TRIGGER WHEN DISTANCE=1 DELAY=-1 DO Schrittmerker_R1Place(10692,10691,FPlace_R1_L6_S4_Check,XPlace_R1_L6_S4_Check) PRIO=-1
;FOLD PTP Place_R1_L6_S4_Check Vel=12 % PPlace_R1_L6_S4_Check Tool[1]:Upper Gripper Base[1]:Rack1;%{PE}%R8.3.21,%MKUKATPBASIS,%CMOVE,%VPTP,%P 1:PTP, 2:Place_R1_L6_S4_Check, 3:, 5:12, 7:PPlace_R1_L6_S4_Check
$BWDSTART=FALSE
PDAT_ACT= PPPlace_R1_L6_S4_Check
FDAT_ACT= FPlace_R1_L6_S4_Check
BAS(#PTP_PARAMS,12)
PTP XPlace_R1_L6_S4_Check
;ENDFOLD

;***************************************************
;FOLD Pruefe Platz frei
IF (DetectPart(CHECK_SHELF,PLACE)==OCCUPIED) THEN
  UP_Rueckzug_R1Place( )
  RETURN
ENDIF
;ENDFOLD
;***************************************************

TRIGGER WHEN DISTANCE=1 DELAY=-1 DO Schrittmerker_R1Place(10693,10692,FPlace_R1_L6_S4_VP3,XPlace_R1_L6_S4_VP3) PRIO=-1
;FOLD LIN Place_R1_L6_S4_VP3 CONT Vel=0.5 m/s LPlace_R1_L6_S4_VP3 Tool[1]:Upper Gripper Base[1]:Rack1;%{PE}%R8.3.21,%MKUKATPBASIS,%CMOVE,%VLIN,%P 1:LIN, 2:Place_R1_L6_S4_VP3, 3:C_DIS C_DIS, 5:0.5, 7:LPlace_R1_L6_S4_VP3
$BWDSTART=FALSE
LDAT_ACT= LLPlace_R1_L6_S4_VP3
FDAT_ACT= FPlace_R1_L6_S4_VP3
BAS(#CP_PARAMS,0.5)
LIN XPlace_R1_L6_S4_VP3 C_DIS C_DIS
;ENDFOLD
TRIGGER WHEN DISTANCE=1 DELAY=-1 DO Schrittmerker_R1Place(10694,10693,FPlace_R1_L6_S4_VP4,XPlace_R1_L6_S4_VP4) PRIO=-1
;FOLD LIN Place_R1_L6_S4_VP4 CONT Vel=0.5 m/s LPlace_R1_L6_S4_VP4 Tool[1]:Upper Gripper Base[1]:Rack1;%{PE}%R8.3.21,%MKUKATPBASIS,%CMOVE,%VLIN,%P 1:LIN, 2:Place_R1_L6_S4_VP4, 3:C_DIS C_DIS, 5:0.5, 7:LPlace_R1_L6_S4_VP4
$BWDSTART=FALSE
LDAT_ACT= LLPlace_R1_L6_S4_VP4
FDAT_ACT= FPlace_R1_L6_S4_VP4
BAS(#CP_PARAMS,0.5)
LIN XPlace_R1_L6_S4_VP4 C_DIS C_DIS
;ENDFOLD
TRIGGER WHEN DISTANCE=1 DELAY=-1 DO Schrittmerker_R1Place(10695,10694,FPlace_R1_L6_S4_VP5,XPlace_R1_L6_S4_VP5) PRIO=-1
;FOLD LIN Place_R1_L6_S4_VP5 CONT Vel=0.5 m/s LPlace_R1_L6_S4_VP5 Tool[1]:Upper Gripper Base[1]:Rack1;%{PE}%R8.3.21,%MKUKATPBASIS,%CMOVE,%VLIN,%P 1:LIN, 2:Place_R1_L6_S4_VP5, 3:C_DIS C_DIS, 5:0.5, 7:LPlace_R1_L6_S4_VP5
$BWDSTART=FALSE
LDAT_ACT= LLPlace_R1_L6_S4_VP5
FDAT_ACT= FPlace_R1_L6_S4_VP5
BAS(#CP_PARAMS,0.5)
LIN XPlace_R1_L6_S4_VP5 C_DIS C_DIS
;ENDFOLD

;FOLD Test the way back home - part 1
CONTINUE
IF ($FLAG[M_Test_GrdstFahren1] AND NOT $FLAG[M_Test_GrdstFahren2]) THEN
  $FLAG[M_Test_GrdstFahren2]=TRUE
  UP_Rueckzug( )
  RETURN
ENDIF
;ENDFOLD

;-------------------------------
; Place part position
;-------------------------------
TRIGGER WHEN DISTANCE=1 DELAY=-1 DO Schrittmerker_R1Place(10696,10697,FPlace_R1_L6_S4_AP,XPlace_R1_L6_S4_AP) PRIO=-1
;FOLD LIN Place_R1_L6_S4_AP Vel=0.2 m/s LPlace_R1_L6_S4_AP Tool[1]:Upper Gripper Base[1]:Rack1;%{PE}%R8.3.21,%MKUKATPBASIS,%CMOVE,%VLIN,%P 1:LIN, 2:Place_R1_L6_S4_AP, 3:, 5:0.2, 7:LPlace_R1_L6_S4_AP
$BWDSTART=FALSE
LDAT_ACT= LLPlace_R1_L6_S4_AP
FDAT_ACT= FPlace_R1_L6_S4_AP
BAS(#CP_PARAMS,0.2)
LIN XPlace_R1_L6_S4_AP
;ENDFOLD

;FOLD Test the way back home - part 2
CONTINUE
IF $FLAG[M_Test_GrdstFahren2] THEN
  $FLAG[M_Test_GrdstFahren2]=FALSE
  UP_Rueckzug( )
  RETURN
ENDIF
;ENDFOLD

;***************************************************
; Disable part lost detection
SetPartLostDetection(NO_PART)
;***************************************************

TRIGGER WHEN DISTANCE=1 DELAY=-1 DO Schrittmerker_R1Place(10697,10698,FPlace_R1_L6_S4_NP1,XPlace_R1_L6_S4_NP1) PRIO=-1
;FOLD LIN Place_R1_L6_S4_NP1 Vel=0.2 m/s LPlace_R1_L6_S4_NP1 Tool[1]:Upper Gripper Base[1]:Rack1;%{PE}%R8.3.21,%MKUKATPBASIS,%CMOVE,%VLIN,%P 1:LIN, 2:Place_R1_L6_S4_NP1, 3:C_DIS C_DIS, 5:0.2, 7:LPlace_R1_L6_S4_NP1
$BWDSTART=FALSE
LDAT_ACT= LLPlace_R1_L6_S4_NP1
FDAT_ACT= FPlace_R1_L6_S4_NP1
BAS(#CP_PARAMS,0.2)
LIN XPlace_R1_L6_S4_NP1
;ENDFOLD

;***************************************************
; Check for part present (empty gripper)
CheckPartPresent(EMPTY_GRIPPER)
;***************************************************
; set load data
SetLoadData( )
;***************************************************

TRIGGER WHEN DISTANCE=1 DELAY=-1 DO Schrittmerker_R1Place(10698,10699,FPlace_R1_L6_S4_NP2,XPlace_R1_L6_S4_NP2) PRIO=-1
;FOLD LIN Place_R1_L6_S4_NP2 CONT Vel=0.5 m/s LPlace_R1_L6_S4_NP2 Tool[1]:Upper Gripper Base[1]:Rack1;%{PE}%R8.3.21,%MKUKATPBASIS,%CMOVE,%VLIN,%P 1:LIN, 2:Place_R1_L6_S4_NP2, 3:C_DIS C_DIS, 5:0.5, 7:LPlace_R1_L6_S4_NP2
$BWDSTART=FALSE
LDAT_ACT= LLPlace_R1_L6_S4_NP2
FDAT_ACT= FPlace_R1_L6_S4_NP2
BAS(#CP_PARAMS,0.5)
LIN XPlace_R1_L6_S4_NP2 C_DIS C_DIS
;ENDFOLD
TRIGGER WHEN DISTANCE=1 DELAY=-1 DO Schrittmerker_R1Place(10699,10700,FPlace_R1_L6_S4_NP3,XPlace_R1_L6_S4_NP3) PRIO=-1
;FOLD LIN Place_R1_L6_S4_NP3 Vel=0.5 m/s LPlace_R1_L6_S4_NP3 Tool[1]:Upper Gripper Base[1]:Rack1;%{PE}%R8.3.21,%MKUKATPBASIS,%CMOVE,%VLIN,%P 1:LIN, 2:Place_R1_L6_S4_NP3, 3:, 5:0.5, 7:LPlace_R1_L6_S4_NP3
$BWDSTART=FALSE
LDAT_ACT= LLPlace_R1_L6_S4_NP3
FDAT_ACT= FPlace_R1_L6_S4_NP3
BAS(#CP_PARAMS,0.5)
LIN XPlace_R1_L6_S4_NP3
;ENDFOLD
TRIGGER WHEN DISTANCE=1 DELAY=-1 DO Schrittmerker_R1Place(10700,10701,FPlace_R1_L6_S4_NP4,XPlace_R1_L6_S4_NP4) PRIO=-1
;FOLD PTP Place_R1_L6_S4_NP4 CONT Vel=100 % PPlace_R1_L6_S4_NP4 Tool[1]:Upper Gripper Base[0];%{PE}%R8.3.21,%MKUKATPBASIS,%CMOVE,%VPTP,%P 1:PTP, 2:Place_R1_L6_S4_NP4, 3:C_DIS, 5:100, 7:PPlace_R1_L6_S4_NP4
$BWDSTART=FALSE
PDAT_ACT= PPPlace_R1_L6_S4_NP4
FDAT_ACT= FPlace_R1_L6_S4_NP4
BAS(#PTP_PARAMS,100)
PTP XPlace_R1_L6_S4_NP4 C_DIS
;ENDFOLD
TRIGGER WHEN DISTANCE=1 DELAY=-1 DO Schrittmerker_R1Place(10701,10702,FPlace_R1_L6_S4_NP5,XPlace_R1_L6_S4_NP5) PRIO=-1
;FOLD PTP Place_R1_L6_S4_NP5 CONT Vel=100 % PPlace_R1_L6_S4_NP5 Tool[1]:Upper Gripper Base[0];%{PE}%R8.3.21,%MKUKATPBASIS,%CMOVE,%VPTP,%P 1:PTP, 2:Place_R1_L6_S4_NP5, 3:C_DIS, 5:100, 7:PPlace_R1_L6_S4_NP5
$BWDSTART=FALSE
PDAT_ACT= PPPlace_R1_L6_S4_NP5
FDAT_ACT= FPlace_R1_L6_S4_NP5
BAS(#PTP_PARAMS,100)
PTP XPlace_R1_L6_S4_NP5 C_DIS
;ENDFOLD
TRIGGER WHEN DISTANCE=1 DELAY=-1 DO Schrittmerker_R1Place(10702,10703,FPlace_R1_L6_S4_NP6,XPlace_R1_L6_S4_NP6) PRIO=-1
;FOLD PTP Place_R1_L6_S4_NP6 CONT Vel=100 % PPlace_R1_L6_S4_NP6 Tool[1]:Upper Gripper Base[0];%{PE}%R8.3.21,%MKUKATPBASIS,%CMOVE,%VPTP,%P 1:PTP, 2:Place_R1_L6_S4_NP6, 3:C_DIS, 5:100, 7:PPlace_R1_L6_S4_NP6
$BWDSTART=FALSE
PDAT_ACT= PPPlace_R1_L6_S4_NP6
FDAT_ACT= FPlace_R1_L6_S4_NP6
BAS(#PTP_PARAMS,100)
PTP XPlace_R1_L6_S4_NP6 C_DIS
;ENDFOLD

TRIGGER WHEN DISTANCE=1 DELAY=-1 DO Schrittmerker_R1Place(10703,10501,FHOME,$nullframe,XHOME) PRIO=-1
;FOLD PTP HOME Vel=100 % PHome;%{PE}%R8.3.21,%MKUKATPBASIS,%CMOVE,%VPTP,%P 1:PTP, 2:HOME, 3:, 5:100, 7:PHome
$BWDSTART=FALSE
PDAT_ACT= PPHome
FDAT_ACT= FHOME
BAS(#PTP_PARAMS,100)
PTP XHOME
;ENDFOLD

;***************************************************
;FOLD Final tasks.
; Robot out of area Rack 1 Level 6
RobAusStorage1_6_A72=RESET_IN_AREA
;***************************************************
; stop cyclic clearence check
$CYCFLAG[ciFreigabeSPS]=DISABLE_MONITORING
;***************************************************
; Disable collision detection
;FOLD COLLDETECT Off ;%{PE}
;FOLD Parameters ;%{h}
;Params IlfProvider=kukaroboter.basistech.inlineforms.colldetect.off; CollDetect.Command=Off
;ENDFOLD
USE_CD_PARAMS(0)
;ENDFOLD
;***************************************************
;ENDFOLD
;***************************************************

END

; ##################################################

GLOBAL DEF UP_Place_R1_L7_S1( )
;***************************************************
; Place part on:
;    Rack  1
;    Level 7
;    Shelf 1
;  RBG Kollision beachten!
;***************************************************
;FOLD Preconditions - Vorraussetzungen
;***************************************************
; Enable collision detection
;FOLD COLLDETECT SetLimits Axis1: 150 % Axis2: 200 % Axis3: 150 % Axis4: 200 % Axis5: 150 % Axis6: 150 % ;%{PE}
;FOLD Parameters ;%{h}
;Params IlfProvider=kukaroboter.basistech.inlineforms.colldetect.setlimits; CollDetect.Command=SetLimits; CollDetect.Axis1=150; CollDetect.Axis2=200; CollDetect.Axis3=150; CollDetect.Axis4=200; CollDetect.Axis5=150; CollDetect.Axis6=150
;ENDFOLD
SET_TQ_VALUES(150, 200, 150, 200, 150, 150)
;ENDFOLD
;***************************************************
; Check for part in gripper (tool 1).
CheckPartPresent(OCCUPIED_GRIPPER,PART_ON_TOOL_1)
;***************************************************
; Enable part lost detection for tool 1
SetPartLostDetection(PART_ON_TOOL_1)
;***************************************************
; Set load data.
SetLoadData( )
;***************************************************
; Robot has to start from home position.
IF NOT $IN_HOME THEN
  UP_HomeToHome(0)
ENDIF
;***************************************************
;ENDFOLD

TRIGGER WHEN DISTANCE=1 DELAY=-1 DO Schrittmerker_R1Place(10501,10501,FHOME,$nullframe,XHOME) PRIO=-1
;FOLD PTP HOME Vel=12 % PHome;%{PE}%R8.3.21,%MKUKATPBASIS,%CMOVE,%VPTP,%P 1:PTP, 2:HOME, 3:, 5:12, 7:PHome
$BWDSTART=FALSE
PDAT_ACT= PPHome
FDAT_ACT= FHOME
BAS(#PTP_PARAMS,12)
PTP XHOME
;ENDFOLD

;***************************************************
;FOLD Area clearence handshake.
IF NOT $FLAG[M_Inbetriebnahme] THEN
  ;-------------------------------------------------
  ; Request area clearence.
  AnfStoer_Store1_7_A105=SET_REQUEST
  ;-------------------------------------------------
  ; Wait for area clearence from PLC.
  WAIT_FOR_INPUT("Frg_Storage1_7_E73",TRUE)
  ;-------------------------------------------------
  ; Reset area clearence request.
  AnfStoer_Store1_7_A105=RESET_REQUEST
  ;-------------------------------------------------
  ; start cyclic clearence check
  $CYCFLAG[ciFreigabeSPS]=Frg_Storage1_7_E73
  ;-------------------------------------------------
ENDIF
;***************************************************
; set "robot in area"
RobAusStorage1_7_A73=SET_IN_AREA
;ENDFOLD
;***************************************************

;***************************************************
;FOLD Check for Teachmode
IF $FLAG[M_Teachen] THEN
  WAIT FOR $T1
ENDIF
;ENDFOLD
;***************************************************

; move to the rack
TRIGGER WHEN DISTANCE=1 DELAY=-1 DO Schrittmerker_R1Place(10710,10501,FPlace_R1_L7_S1_VP1,XPlace_R1_L7_S1_VP1) PRIO=-1
;FOLD PTP Place_R1_L7_S1_VP1 CONT Vel=12 % PPlace_R1_L7_S1_VP1 Tool[1]:Upper Gripper Base[0];%{PE}%R8.3.21,%MKUKATPBASIS,%CMOVE,%VPTP,%P 1:PTP, 2:Place_R1_L7_S1_VP1, 3:C_DIS, 5:12, 7:PPlace_R1_L7_S1_VP1
$BWDSTART=FALSE
PDAT_ACT= PPPlace_R1_L7_S1_VP1
FDAT_ACT= FPlace_R1_L7_S1_VP1
BAS(#PTP_PARAMS,12)
PTP XPlace_R1_L7_S1_VP1 C_DIS
;ENDFOLD
TRIGGER WHEN DISTANCE=1 DELAY=-1 DO Schrittmerker_R1Place(10711,10710,FPlace_R1_L7_S1_VP2,XPlace_R1_L7_S1_VP2) PRIO=-1
;FOLD PTP Place_R1_L7_S1_VP2 CONT Vel=12 % PPlace_R1_L7_S1_VP2 Tool[1]:Upper Gripper Base[0];%{PE}%R8.3.21,%MKUKATPBASIS,%CMOVE,%VPTP,%P 1:PTP, 2:Place_R1_L7_S1_VP2, 3:C_DIS, 5:12, 7:PPlace_R1_L7_S1_VP2
$BWDSTART=FALSE
PDAT_ACT= PPPlace_R1_L7_S1_VP2
FDAT_ACT= FPlace_R1_L7_S1_VP2
BAS(#PTP_PARAMS,12)
PTP XPlace_R1_L7_S1_VP2 C_DIS
;ENDFOLD
TRIGGER WHEN DISTANCE=1 DELAY=-1 DO Schrittmerker_R1Place(10712,10711,FPlace_R1_L7_S1_VP3,XPlace_R1_L7_S1_VP3) PRIO=-1
;FOLD PTP Place_R1_L7_S1_VP3 CONT Vel=12 % PPlace_R1_L7_S1_VP3 Tool[1]:Upper Gripper Base[0];%{PE}%R8.3.21,%MKUKATPBASIS,%CMOVE,%VPTP,%P 1:PTP, 2:Place_R1_L7_S1_VP3, 3:C_DIS, 5:12, 7:PPlace_R1_L7_S1_VP3
$BWDSTART=FALSE
PDAT_ACT= PPPlace_R1_L7_S1_VP3
FDAT_ACT= FPlace_R1_L7_S1_VP3
BAS(#PTP_PARAMS,12)
PTP XPlace_R1_L7_S1_VP3 C_DIS
;ENDFOLD
TRIGGER WHEN DISTANCE=1 DELAY=-1 DO Schrittmerker_R1Place(10713,10712,FPlace_R1_L7_S1_VP4,XPlace_R1_L7_S1_VP4) PRIO=-1
;FOLD PTP Place_R1_L7_S1_VP4 CONT Vel=12 % PPlace_R1_L7_S1_VP4 Tool[1]:Upper Gripper Base[0];%{PE}%R8.3.21,%MKUKATPBASIS,%CMOVE,%VPTP,%P 1:PTP, 2:Place_R1_L7_S1_VP4, 3:C_DIS, 5:12, 7:PPlace_R1_L7_S1_VP4
$BWDSTART=FALSE
PDAT_ACT= PPPlace_R1_L7_S1_VP4
FDAT_ACT= FPlace_R1_L7_S1_VP4
BAS(#PTP_PARAMS,12)
PTP XPlace_R1_L7_S1_VP4 C_DIS
;ENDFOLD
TRIGGER WHEN DISTANCE=1 DELAY=-1 DO Schrittmerker_R1Place(10714,10713,FPlace_R1_L7_S1_VP5,XPlace_R1_L7_S1_VP5) PRIO=-1
;FOLD PTP Place_R1_L7_S1_VP5 CONT Vel=12 % PPlace_R1_L7_S1_VP5 Tool[1]:Upper Gripper Base[0];%{PE}%R8.3.21,%MKUKATPBASIS,%CMOVE,%VPTP,%P 1:PTP, 2:Place_R1_L7_S1_VP5, 3:C_DIS, 5:12, 7:PPlace_R1_L7_S1_VP5
$BWDSTART=FALSE
PDAT_ACT= PPPlace_R1_L7_S1_VP5
FDAT_ACT= FPlace_R1_L7_S1_VP5
BAS(#PTP_PARAMS,12)
PTP XPlace_R1_L7_S1_VP5 C_DIS
;ENDFOLD
TRIGGER WHEN DISTANCE=1 DELAY=-1 DO Schrittmerker_R1Place(10715,10714,FPlace_R1_L7_S1_VP6,XPlace_R1_L7_S1_VP6) PRIO=-1
;FOLD PTP Place_R1_L7_S1_VP6 CONT Vel=12 % PPlace_R1_L7_S1_VP6 Tool[1]:Upper Gripper Base[0];%{PE}%R8.3.21,%MKUKATPBASIS,%CMOVE,%VPTP,%P 1:PTP, 2:Place_R1_L7_S1_VP6, 3:C_DIS, 5:12, 7:PPlace_R1_L7_S1_VP6
$BWDSTART=FALSE
PDAT_ACT= PPPlace_R1_L7_S1_VP6
FDAT_ACT= FPlace_R1_L7_S1_VP6
BAS(#PTP_PARAMS,12)
PTP XPlace_R1_L7_S1_VP6 C_DIS
;ENDFOLD
TRIGGER WHEN DISTANCE=1 DELAY=-1 DO Schrittmerker_R1Place(10716,10715,FPlace_R1_L7_S1_VP7,XPlace_R1_L7_S1_VP7) PRIO=-1
;FOLD PTP Place_R1_L7_S1_VP7 CONT Vel=12 % PPlace_R1_L7_S1_VP7 Tool[1]:Upper Gripper Base[0];%{PE}%R8.3.21,%MKUKATPBASIS,%CMOVE,%VPTP,%P 1:PTP, 2:Place_R1_L7_S1_VP7, 3:C_DIS, 5:12, 7:PPlace_R1_L7_S1_VP7
$BWDSTART=FALSE
PDAT_ACT= PPPlace_R1_L7_S1_VP7
FDAT_ACT= FPlace_R1_L7_S1_VP7
BAS(#PTP_PARAMS,12)
PTP XPlace_R1_L7_S1_VP7 C_DIS
;ENDFOLD
TRIGGER WHEN DISTANCE=1 DELAY=-1 DO Schrittmerker_R1Place(10717,10716,FPlace_R1_L7_S1_VP8,XPlace_R1_L7_S1_VP8) PRIO=-1
;FOLD PTP Place_R1_L7_S1_VP8 CONT Vel=12 % PPlace_R1_L7_S1_VP8 Tool[1]:Upper Gripper Base[1]:Rack1;%{PE}%R8.3.21,%MKUKATPBASIS,%CMOVE,%VPTP,%P 1:PTP, 2:Place_R1_L7_S1_VP8, 3:C_DIS, 5:12, 7:PPlace_R1_L7_S1_VP8
$BWDSTART=FALSE
PDAT_ACT= PPPlace_R1_L7_S1_VP8
FDAT_ACT= FPlace_R1_L7_S1_VP8
BAS(#PTP_PARAMS,12)
PTP XPlace_R1_L7_S1_VP8 C_DIS
;ENDFOLD

TRIGGER WHEN DISTANCE=1 DELAY=-1 DO Schrittmerker_R1Place(10718,10717,FPlace_R1_L7_S1_Check,XPlace_R1_L7_S1_Check) PRIO=-1
;FOLD PTP Place_R1_L7_S1_Check Vel=12 % PPlace_R1_L7_S1_Check Tool[1]:Upper Gripper Base[1]:Rack1;%{PE}%R8.3.21,%MKUKATPBASIS,%CMOVE,%VPTP,%P 1:PTP, 2:Place_R1_L7_S1_Check, 3:, 5:12, 7:PPlace_R1_L7_S1_Check
$BWDSTART=FALSE
PDAT_ACT= PPPlace_R1_L7_S1_Check
FDAT_ACT= FPlace_R1_L7_S1_Check
BAS(#PTP_PARAMS,12)
PTP XPlace_R1_L7_S1_Check
;ENDFOLD

;***************************************************
;FOLD Pruefe Platz frei
IF (DetectPart(CHECK_SHELF,PLACE)==OCCUPIED) THEN
  UP_Rueckzug_R1Place( )
  RETURN
ENDIF
;ENDFOLD
;***************************************************

TRIGGER WHEN DISTANCE=1 DELAY=-1 DO Schrittmerker_R1Place(10719,10718,FPlace_R1_L7_S1_VP9,XPlace_R1_L7_S1_VP9) PRIO=-1
;FOLD LIN Place_R1_L7_S1_VP9 CONT Vel=0.5 m/s LPlace_R1_L7_S1_VP9 Tool[1]:Upper Gripper Base[1]:Rack1;%{PE}%R8.3.21,%MKUKATPBASIS,%CMOVE,%VLIN,%P 1:LIN, 2:Place_R1_L7_S1_VP9, 3:C_DIS C_DIS, 5:0.5, 7:LPlace_R1_L7_S1_VP9
$BWDSTART=FALSE
LDAT_ACT= LLPlace_R1_L7_S1_VP9
FDAT_ACT= FPlace_R1_L7_S1_VP9
BAS(#CP_PARAMS,0.5)
LIN XPlace_R1_L7_S1_VP9 C_DIS C_DIS
;ENDFOLD
TRIGGER WHEN DISTANCE=1 DELAY=-1 DO Schrittmerker_R1Place(10720,10719,FPlace_R1_L7_S1_VP10,XPlace_R1_L7_S1_VP10) PRIO=-1
;FOLD LIN Place_R1_L7_S1_VP10 CONT Vel=0.5 m/s LPlace_R1_L7_S1_VP10 Tool[1]:Upper Gripper Base[1]:Rack1;%{PE}%R8.3.21,%MKUKATPBASIS,%CMOVE,%VLIN,%P 1:LIN, 2:Place_R1_L7_S1_VP10, 3:C_DIS C_DIS, 5:0.5, 7:LPlace_R1_L7_S1_VP10
$BWDSTART=FALSE
LDAT_ACT= LLPlace_R1_L7_S1_VP10
FDAT_ACT= FPlace_R1_L7_S1_VP10
BAS(#CP_PARAMS,0.5)
LIN XPlace_R1_L7_S1_VP10 C_DIS C_DIS
;ENDFOLD
TRIGGER WHEN DISTANCE=1 DELAY=-1 DO Schrittmerker_R1Place(10721,10720,FPlace_R1_L7_S1_VP11,XPlace_R1_L7_S1_VP11) PRIO=-1
;FOLD LIN Place_R1_L7_S1_VP11 CONT Vel=0.5 m/s LPlace_R1_L7_S1_VP11 Tool[1]:Upper Gripper Base[1]:Rack1;%{PE}%R8.3.21,%MKUKATPBASIS,%CMOVE,%VLIN,%P 1:LIN, 2:Place_R1_L7_S1_VP11, 3:C_DIS C_DIS, 5:0.5, 7:LPlace_R1_L7_S1_VP11
$BWDSTART=FALSE
LDAT_ACT= LLPlace_R1_L7_S1_VP11
FDAT_ACT= FPlace_R1_L7_S1_VP11
BAS(#CP_PARAMS,0.5)
LIN XPlace_R1_L7_S1_VP11 C_DIS C_DIS
;ENDFOLD

;FOLD Test the way back home - part 1
CONTINUE
IF ($FLAG[M_Test_GrdstFahren1] AND NOT $FLAG[M_Test_GrdstFahren2]) THEN
  $FLAG[M_Test_GrdstFahren2]=TRUE
  UP_Rueckzug( )
  RETURN
ENDIF
;ENDFOLD

;-------------------------------
; Place part position
;-------------------------------
TRIGGER WHEN DISTANCE=1 DELAY=-1 DO Schrittmerker_R1Place(10722,10723,FPlace_R1_L7_S1_AP,XPlace_R1_L7_S1_AP) PRIO=-1
;FOLD LIN Place_R1_L7_S1_AP Vel=0.2 m/s LPlace_R1_L7_S1_AP Tool[1]:Upper Gripper Base[1]:Rack1;%{PE}%R8.3.21,%MKUKATPBASIS,%CMOVE,%VLIN,%P 1:LIN, 2:Place_R1_L7_S1_AP, 3:, 5:0.2, 7:LPlace_R1_L7_S1_AP
$BWDSTART=FALSE
LDAT_ACT= LLPlace_R1_L7_S1_AP
FDAT_ACT= FPlace_R1_L7_S1_AP
BAS(#CP_PARAMS,0.2)
LIN XPlace_R1_L7_S1_AP
;ENDFOLD

;FOLD Test the way back home - part 2
CONTINUE
IF $FLAG[M_Test_GrdstFahren2] THEN
  $FLAG[M_Test_GrdstFahren2]=FALSE
  UP_Rueckzug( )
  RETURN
ENDIF
;ENDFOLD

;***************************************************
; Disable part lost detection
SetPartLostDetection(NO_PART)
;***************************************************

TRIGGER WHEN DISTANCE=1 DELAY=-1 DO Schrittmerker_R1Place(10723,10724,FPlace_R1_L7_S1_NP1,XPlace_R1_L7_S1_NP1) PRIO=-1
;FOLD LIN Place_R1_L7_S1_NP1 Vel=0.2 m/s LPlace_R1_L7_S1_NP1 Tool[1]:Upper Gripper Base[1]:Rack1;%{PE}%R8.3.21,%MKUKATPBASIS,%CMOVE,%VLIN,%P 1:LIN, 2:Place_R1_L7_S1_NP1, 3:C_DIS C_DIS, 5:0.2, 7:LPlace_R1_L7_S1_NP1
$BWDSTART=FALSE
LDAT_ACT= LLPlace_R1_L7_S1_NP1
FDAT_ACT= FPlace_R1_L7_S1_NP1
BAS(#CP_PARAMS,0.2)
LIN XPlace_R1_L7_S1_NP1
;ENDFOLD

;***************************************************
; Check for part present (empty gripper)
CheckPartPresent(EMPTY_GRIPPER)
;***************************************************
; set load data
SetLoadData( )
;***************************************************

TRIGGER WHEN DISTANCE=1 DELAY=-1 DO Schrittmerker_R1Place(10724,10725,FPlace_R1_L7_S1_NP2,XPlace_R1_L7_S1_NP2) PRIO=-1
;FOLD LIN Place_R1_L7_S1_NP2 CONT Vel=0.5 m/s LPlace_R1_L7_S1_NP2 Tool[1]:Upper Gripper Base[1]:Rack1;%{PE}%R8.3.21,%MKUKATPBASIS,%CMOVE,%VLIN,%P 1:LIN, 2:Place_R1_L7_S1_NP2, 3:C_DIS C_DIS, 5:0.5, 7:LPlace_R1_L7_S1_NP2
$BWDSTART=FALSE
LDAT_ACT= LLPlace_R1_L7_S1_NP2
FDAT_ACT= FPlace_R1_L7_S1_NP2
BAS(#CP_PARAMS,0.5)
LIN XPlace_R1_L7_S1_NP2 C_DIS C_DIS
;ENDFOLD
TRIGGER WHEN DISTANCE=1 DELAY=-1 DO Schrittmerker_R1Place(10725,10726,FPlace_R1_L7_S1_NP3,XPlace_R1_L7_S1_NP3) PRIO=-1
;FOLD LIN Place_R1_L7_S1_NP3 Vel=0.5 m/s LPlace_R1_L7_S1_NP3 Tool[1]:Upper Gripper Base[1]:Rack1;%{PE}%R8.3.21,%MKUKATPBASIS,%CMOVE,%VLIN,%P 1:LIN, 2:Place_R1_L7_S1_NP3, 3:, 5:0.5, 7:LPlace_R1_L7_S1_NP3
$BWDSTART=FALSE
LDAT_ACT= LLPlace_R1_L7_S1_NP3
FDAT_ACT= FPlace_R1_L7_S1_NP3
BAS(#CP_PARAMS,0.5)
LIN XPlace_R1_L7_S1_NP3
;ENDFOLD
TRIGGER WHEN DISTANCE=1 DELAY=-1 DO Schrittmerker_R1Place(10726,10727,FPlace_R1_L7_S1_NP4,XPlace_R1_L7_S1_NP4) PRIO=-1
;FOLD PTP Place_R1_L7_S1_NP4 CONT Vel=100 % PPlace_R1_L7_S1_NP4 Tool[1]:Upper Gripper Base[1]:Rack1;%{PE}%R8.3.21,%MKUKATPBASIS,%CMOVE,%VPTP,%P 1:PTP, 2:Place_R1_L7_S1_NP4, 3:C_DIS, 5:100, 7:PPlace_R1_L7_S1_NP4
$BWDSTART=FALSE
PDAT_ACT= PPPlace_R1_L7_S1_NP4
FDAT_ACT= FPlace_R1_L7_S1_NP4
BAS(#PTP_PARAMS,100)
PTP XPlace_R1_L7_S1_NP4 C_DIS
;ENDFOLD
TRIGGER WHEN DISTANCE=1 DELAY=-1 DO Schrittmerker_R1Place(10727,10728,FPlace_R1_L7_S1_NP5,XPlace_R1_L7_S1_NP5) PRIO=-1
;FOLD PTP Place_R1_L7_S1_NP5 CONT Vel=100 % PPlace_R1_L7_S1_NP5 Tool[1]:Upper Gripper Base[0];%{PE}%R8.3.21,%MKUKATPBASIS,%CMOVE,%VPTP,%P 1:PTP, 2:Place_R1_L7_S1_NP5, 3:C_DIS, 5:100, 7:PPlace_R1_L7_S1_NP5
$BWDSTART=FALSE
PDAT_ACT= PPPlace_R1_L7_S1_NP5
FDAT_ACT= FPlace_R1_L7_S1_NP5
BAS(#PTP_PARAMS,100)
PTP XPlace_R1_L7_S1_NP5 C_DIS
;ENDFOLD
TRIGGER WHEN DISTANCE=1 DELAY=-1 DO Schrittmerker_R1Place(10728,10729,FPlace_R1_L7_S1_NP6,XPlace_R1_L7_S1_NP6) PRIO=-1
;FOLD PTP Place_R1_L7_S1_NP6 CONT Vel=100 % PPlace_R1_L7_S1_NP6 Tool[1]:Upper Gripper Base[0];%{PE}%R8.3.21,%MKUKATPBASIS,%CMOVE,%VPTP,%P 1:PTP, 2:Place_R1_L7_S1_NP6, 3:C_DIS, 5:100, 7:PPlace_R1_L7_S1_NP6
$BWDSTART=FALSE
PDAT_ACT= PPPlace_R1_L7_S1_NP6
FDAT_ACT= FPlace_R1_L7_S1_NP6
BAS(#PTP_PARAMS,100)
PTP XPlace_R1_L7_S1_NP6 C_DIS
;ENDFOLD
TRIGGER WHEN DISTANCE=1 DELAY=-1 DO Schrittmerker_R1Place(10729,10730,FPlace_R1_L7_S1_NP7,XPlace_R1_L7_S1_NP7) PRIO=-1
;FOLD PTP Place_R1_L7_S1_NP7 CONT Vel=100 % PPlace_R1_L7_S1_NP7 Tool[1]:Upper Gripper Base[0];%{PE}%R8.3.21,%MKUKATPBASIS,%CMOVE,%VPTP,%P 1:PTP, 2:Place_R1_L7_S1_NP7, 3:C_DIS, 5:100, 7:PPlace_R1_L7_S1_NP7
$BWDSTART=FALSE
PDAT_ACT= PPPlace_R1_L7_S1_NP7
FDAT_ACT= FPlace_R1_L7_S1_NP7
BAS(#PTP_PARAMS,100)
PTP XPlace_R1_L7_S1_NP7 C_DIS
;ENDFOLD

TRIGGER WHEN DISTANCE=1 DELAY=-1 DO Schrittmerker_R1Place(10730,10501,FHOME,$nullframe,XHOME) PRIO=-1
;FOLD PTP HOME Vel=100 % PHome;%{PE}%R8.3.21,%MKUKATPBASIS,%CMOVE,%VPTP,%P 1:PTP, 2:HOME, 3:, 5:100, 7:PHome
$BWDSTART=FALSE
PDAT_ACT= PPHome
FDAT_ACT= FHOME
BAS(#PTP_PARAMS,100)
PTP XHOME
;ENDFOLD

;***************************************************
;FOLD Final tasks.
; Robot out of area Rack 1 Level 7
RobAusStorage1_7_A73=RESET_IN_AREA
;***************************************************
; stop cyclic clearence check
$CYCFLAG[ciFreigabeSPS]=DISABLE_MONITORING
;***************************************************
; Disable collision detection
;FOLD COLLDETECT Off ;%{PE}
;FOLD Parameters ;%{h}
;Params IlfProvider=kukaroboter.basistech.inlineforms.colldetect.off; CollDetect.Command=Off
;ENDFOLD
USE_CD_PARAMS(0)
;ENDFOLD
;***************************************************
;ENDFOLD
;***************************************************

END

; ##################################################

GLOBAL DEF UP_Place_R1_L7_S2( )
;***************************************************
; Place part on:
;    Rack  1
;    Level 7
;    Shelf 2
;***************************************************
;FOLD Preconditions - Vorraussetzungen
;***************************************************
; Enable collision detection
;FOLD COLLDETECT SetLimits Axis1: 150 % Axis2: 200 % Axis3: 150 % Axis4: 200 % Axis5: 150 % Axis6: 150 % ;%{PE}
;FOLD Parameters ;%{h}
;Params IlfProvider=kukaroboter.basistech.inlineforms.colldetect.setlimits; CollDetect.Command=SetLimits; CollDetect.Axis1=150; CollDetect.Axis2=200; CollDetect.Axis3=150; CollDetect.Axis4=200; CollDetect.Axis5=150; CollDetect.Axis6=150
;ENDFOLD
SET_TQ_VALUES(150, 200, 150, 200, 150, 150)
;ENDFOLD
;***************************************************
; Check for part in gripper (tool 1).
CheckPartPresent(OCCUPIED_GRIPPER,PART_ON_TOOL_1)
;***************************************************
; Enable part lost detection for tool 1
SetPartLostDetection(PART_ON_TOOL_1)
;***************************************************
; Set load data.
SetLoadData( )
;***************************************************
; Robot has to start from home position.
IF NOT $IN_HOME THEN
  UP_HomeToHome(0)
ENDIF
;***************************************************
;ENDFOLD

TRIGGER WHEN DISTANCE=1 DELAY=-1 DO Schrittmerker_R1Place(10501,10501,FHOME,$nullframe,XHOME) PRIO=-1
;FOLD PTP HOME Vel=12 % PHome;%{PE}%R8.3.21,%MKUKATPBASIS,%CMOVE,%VPTP,%P 1:PTP, 2:HOME, 3:, 5:12, 7:PHome
$BWDSTART=FALSE
PDAT_ACT= PPHome
FDAT_ACT= FHOME
BAS(#PTP_PARAMS,12)
PTP XHOME
;ENDFOLD

;***************************************************
;FOLD Area clearence handshake.
IF NOT $FLAG[M_Inbetriebnahme] THEN
  ;-------------------------------------------------
  ; Request area clearence.
  AnfStoer_Store1_7_A105=SET_REQUEST
  ;-------------------------------------------------
  ; Wait for area clearence from PLC.
  WAIT_FOR_INPUT("Frg_Storage1_7_E73",TRUE)
  ;-------------------------------------------------
  ; Reset area clearence request.
  AnfStoer_Store1_7_A105=RESET_REQUEST
  ;-------------------------------------------------
  ; start cyclic clearence check
  $CYCFLAG[ciFreigabeSPS]=Frg_Storage1_7_E73
  ;-------------------------------------------------
ENDIF
;***************************************************
; set "robot in area"
RobAusStorage1_7_A73=SET_IN_AREA
;ENDFOLD
;***************************************************

;***************************************************
;FOLD Check for Teachmode
IF $FLAG[M_Teachen] THEN
  WAIT FOR $T1
ENDIF
;ENDFOLD
;***************************************************

; move to the rack
TRIGGER WHEN DISTANCE=1 DELAY=-1 DO Schrittmerker_R1Place(10740,10501,FPlace_R1_L7_S2_VP1,XPlace_R1_L7_S2_VP1) PRIO=-1
;FOLD PTP Place_R1_L7_S2_VP1 CONT Vel=12 % PPlace_R1_L7_S2_VP1 Tool[1]:Upper Gripper Base[0];%{PE}%R8.3.21,%MKUKATPBASIS,%CMOVE,%VPTP,%P 1:PTP, 2:Place_R1_L7_S2_VP1, 3:C_DIS, 5:12, 7:PPlace_R1_L7_S2_VP1
$BWDSTART=FALSE
PDAT_ACT= PPPlace_R1_L7_S2_VP1
FDAT_ACT= FPlace_R1_L7_S2_VP1
BAS(#PTP_PARAMS,12)
PTP XPlace_R1_L7_S2_VP1 C_DIS
;ENDFOLD
TRIGGER WHEN DISTANCE=1 DELAY=-1 DO Schrittmerker_R1Place(10741,10740,FPlace_R1_L7_S2_VP2,XPlace_R1_L7_S2_VP2) PRIO=-1
;FOLD PTP Place_R1_L7_S2_VP2 CONT Vel=12 % PPlace_R1_L7_S2_VP2 Tool[1]:Upper Gripper Base[0];%{PE}%R8.3.21,%MKUKATPBASIS,%CMOVE,%VPTP,%P 1:PTP, 2:Place_R1_L7_S2_VP2, 3:C_DIS, 5:12, 7:PPlace_R1_L7_S2_VP2
$BWDSTART=FALSE
PDAT_ACT= PPPlace_R1_L7_S2_VP2
FDAT_ACT= FPlace_R1_L7_S2_VP2
BAS(#PTP_PARAMS,12)
PTP XPlace_R1_L7_S2_VP2 C_DIS
;ENDFOLD
TRIGGER WHEN DISTANCE=1 DELAY=-1 DO Schrittmerker_R1Place(10742,10741,FPlace_R1_L7_S2_VP3,XPlace_R1_L7_S2_VP3) PRIO=-1
;FOLD PTP Place_R1_L7_S2_VP3 CONT Vel=12 % PPlace_R1_L7_S2_VP3 Tool[1]:Upper Gripper Base[0];%{PE}%R8.3.21,%MKUKATPBASIS,%CMOVE,%VPTP,%P 1:PTP, 2:Place_R1_L7_S2_VP3, 3:C_DIS, 5:12, 7:PPlace_R1_L7_S2_VP3
$BWDSTART=FALSE
PDAT_ACT= PPPlace_R1_L7_S2_VP3
FDAT_ACT= FPlace_R1_L7_S2_VP3
BAS(#PTP_PARAMS,12)
PTP XPlace_R1_L7_S2_VP3 C_DIS
;ENDFOLD
TRIGGER WHEN DISTANCE=1 DELAY=-1 DO Schrittmerker_R1Place(10743,10742,FPlace_R1_L7_S2_VP4,XPlace_R1_L7_S2_VP4) PRIO=-1
;FOLD PTP Place_R1_L7_S2_VP4 CONT Vel=12 % PPlace_R1_L7_S2_VP4 Tool[1]:Upper Gripper Base[0];%{PE}%R8.3.21,%MKUKATPBASIS,%CMOVE,%VPTP,%P 1:PTP, 2:Place_R1_L7_S2_VP4, 3:C_DIS, 5:12, 7:PPlace_R1_L7_S2_VP4
$BWDSTART=FALSE
PDAT_ACT= PPPlace_R1_L7_S2_VP4
FDAT_ACT= FPlace_R1_L7_S2_VP4
BAS(#PTP_PARAMS,12)
PTP XPlace_R1_L7_S2_VP4 C_DIS
;ENDFOLD
TRIGGER WHEN DISTANCE=1 DELAY=-1 DO Schrittmerker_R1Place(10744,10743,FPlace_R1_L7_S2_VP5,XPlace_R1_L7_S2_VP5) PRIO=-1
;FOLD PTP Place_R1_L7_S2_VP5 CONT Vel=12 % PPlace_R1_L7_S2_VP5 Tool[1]:Upper Gripper Base[0];%{PE}%R8.3.21,%MKUKATPBASIS,%CMOVE,%VPTP,%P 1:PTP, 2:Place_R1_L7_S2_VP5, 3:C_DIS, 5:12, 7:PPlace_R1_L7_S2_VP5
$BWDSTART=FALSE
PDAT_ACT= PPPlace_R1_L7_S2_VP5
FDAT_ACT= FPlace_R1_L7_S2_VP5
BAS(#PTP_PARAMS,12)
PTP XPlace_R1_L7_S2_VP5 C_DIS
;ENDFOLD
TRIGGER WHEN DISTANCE=1 DELAY=-1 DO Schrittmerker_R1Place(10745,10744,FPlace_R1_L7_S2_VP6,XPlace_R1_L7_S2_VP6) PRIO=-1
;FOLD PTP Place_R1_L7_S2_VP6 CONT Vel=12 % PPlace_R1_L7_S2_VP6 Tool[1]:Upper Gripper Base[0];%{PE}%R8.3.21,%MKUKATPBASIS,%CMOVE,%VPTP,%P 1:PTP, 2:Place_R1_L7_S2_VP6, 3:C_DIS, 5:12, 7:PPlace_R1_L7_S2_VP6
$BWDSTART=FALSE
PDAT_ACT= PPPlace_R1_L7_S2_VP6
FDAT_ACT= FPlace_R1_L7_S2_VP6
BAS(#PTP_PARAMS,12)
PTP XPlace_R1_L7_S2_VP6 C_DIS
;ENDFOLD
TRIGGER WHEN DISTANCE=1 DELAY=-1 DO Schrittmerker_R1Place(10746,10745,FPlace_R1_L7_S2_VP7,XPlace_R1_L7_S2_VP7) PRIO=-1
;FOLD PTP Place_R1_L7_S2_VP7 CONT Vel=12 % PPlace_R1_L7_S2_VP7 Tool[1]:Upper Gripper Base[0];%{PE}%R8.3.21,%MKUKATPBASIS,%CMOVE,%VPTP,%P 1:PTP, 2:Place_R1_L7_S2_VP7, 3:C_DIS, 5:12, 7:PPlace_R1_L7_S2_VP7
$BWDSTART=FALSE
PDAT_ACT= PPPlace_R1_L7_S2_VP7
FDAT_ACT= FPlace_R1_L7_S2_VP7
BAS(#PTP_PARAMS,12)
PTP XPlace_R1_L7_S2_VP7 C_DIS
;ENDFOLD
TRIGGER WHEN DISTANCE=1 DELAY=-1 DO Schrittmerker_R1Place(10747,10746,FPlace_R1_L7_S2_VP8,XPlace_R1_L7_S2_VP8) PRIO=-1
;FOLD PTP Place_R1_L7_S2_VP8 CONT Vel=12 % PPlace_R1_L7_S2_VP8 Tool[1]:Upper Gripper Base[1]:Rack1;%{PE}%R8.3.21,%MKUKATPBASIS,%CMOVE,%VPTP,%P 1:PTP, 2:Place_R1_L7_S2_VP8, 3:C_DIS, 5:12, 7:PPlace_R1_L7_S2_VP8
$BWDSTART=FALSE
PDAT_ACT= PPPlace_R1_L7_S2_VP8
FDAT_ACT= FPlace_R1_L7_S2_VP8
BAS(#PTP_PARAMS,12)
PTP XPlace_R1_L7_S2_VP8 C_DIS
;ENDFOLD

TRIGGER WHEN DISTANCE=1 DELAY=-1 DO Schrittmerker_R1Place(10748,10747,FPlace_R1_L7_S2_Check,XPlace_R1_L7_S2_Check) PRIO=-1
;FOLD PTP Place_R1_L7_S2_Check Vel=12 % PPlace_R1_L7_S2_Check Tool[1]:Upper Gripper Base[1]:Rack1;%{PE}%R8.3.21,%MKUKATPBASIS,%CMOVE,%VPTP,%P 1:PTP, 2:Place_R1_L7_S2_Check, 3:, 5:12, 7:PPlace_R1_L7_S2_Check
$BWDSTART=FALSE
PDAT_ACT= PPPlace_R1_L7_S2_Check
FDAT_ACT= FPlace_R1_L7_S2_Check
BAS(#PTP_PARAMS,12)
PTP XPlace_R1_L7_S2_Check
;ENDFOLD

;***************************************************
;FOLD Pruefe Platz frei
IF (DetectPart(CHECK_SHELF,PLACE)==OCCUPIED) THEN
  UP_Rueckzug_R1Place( )
  RETURN
ENDIF
;ENDFOLD
;***************************************************

TRIGGER WHEN DISTANCE=1 DELAY=-1 DO Schrittmerker_R1Place(10749,10748,FPlace_R1_L7_S2_VP9,XPlace_R1_L7_S2_VP9) PRIO=-1
;FOLD LIN Place_R1_L7_S2_VP9 CONT Vel=0.5 m/s LPlace_R1_L7_S2_VP9 Tool[1]:Upper Gripper Base[1]:Rack1;%{PE}%R8.3.21,%MKUKATPBASIS,%CMOVE,%VLIN,%P 1:LIN, 2:Place_R1_L7_S2_VP9, 3:C_DIS C_DIS, 5:0.5, 7:LPlace_R1_L7_S2_VP9
$BWDSTART=FALSE
LDAT_ACT= LLPlace_R1_L7_S2_VP9
FDAT_ACT= FPlace_R1_L7_S2_VP9
BAS(#CP_PARAMS,0.5)
LIN XPlace_R1_L7_S2_VP9 C_DIS C_DIS
;ENDFOLD
TRIGGER WHEN DISTANCE=1 DELAY=-1 DO Schrittmerker_R1Place(10750,10749,FPlace_R1_L7_S2_VP10,XPlace_R1_L7_S2_VP10) PRIO=-1
;FOLD LIN Place_R1_L7_S2_VP10 CONT Vel=0.5 m/s LPlace_R1_L7_S2_VP10 Tool[1]:Upper Gripper Base[1]:Rack1;%{PE}%R8.3.21,%MKUKATPBASIS,%CMOVE,%VLIN,%P 1:LIN, 2:Place_R1_L7_S2_VP10, 3:C_DIS C_DIS, 5:0.5, 7:LPlace_R1_L7_S2_VP10
$BWDSTART=FALSE
LDAT_ACT= LLPlace_R1_L7_S2_VP10
FDAT_ACT= FPlace_R1_L7_S2_VP10
BAS(#CP_PARAMS,0.5)
LIN XPlace_R1_L7_S2_VP10 C_DIS C_DIS
;ENDFOLD
TRIGGER WHEN DISTANCE=1 DELAY=-1 DO Schrittmerker_R1Place(10751,10750,FPlace_R1_L7_S2_VP11,XPlace_R1_L7_S2_VP11) PRIO=-1
;FOLD LIN Place_R1_L7_S2_VP11 CONT Vel=0.5 m/s LPlace_R1_L7_S2_VP11 Tool[1]:Upper Gripper Base[1]:Rack1;%{PE}%R8.3.21,%MKUKATPBASIS,%CMOVE,%VLIN,%P 1:LIN, 2:Place_R1_L7_S2_VP11, 3:C_DIS C_DIS, 5:0.5, 7:LPlace_R1_L7_S2_VP11
$BWDSTART=FALSE
LDAT_ACT= LLPlace_R1_L7_S2_VP11
FDAT_ACT= FPlace_R1_L7_S2_VP11
BAS(#CP_PARAMS,0.5)
LIN XPlace_R1_L7_S2_VP11 C_DIS C_DIS
;ENDFOLD
TRIGGER WHEN DISTANCE=1 DELAY=-1 DO Schrittmerker_R1Place(10752,10751,FPlace_R1_L7_S2_VP12,XPlace_R1_L7_S2_VP12) PRIO=-1
;FOLD LIN Place_R1_L7_S2_VP12 CONT Vel=0.5 m/s LPlace_R1_L7_S2_VP12 Tool[1]:Upper Gripper Base[1]:Rack1;%{PE}%R8.3.21,%MKUKATPBASIS,%CMOVE,%VLIN,%P 1:LIN, 2:Place_R1_L7_S2_VP12, 3:C_DIS C_DIS, 5:0.5, 7:LPlace_R1_L7_S2_VP12
$BWDSTART=FALSE
LDAT_ACT= LLPlace_R1_L7_S2_VP12
FDAT_ACT= FPlace_R1_L7_S2_VP12
BAS(#CP_PARAMS,0.5)
LIN XPlace_R1_L7_S2_VP12 C_DIS C_DIS
;ENDFOLD

;FOLD Test the way back home - part 1
CONTINUE
IF ($FLAG[M_Test_GrdstFahren1] AND NOT $FLAG[M_Test_GrdstFahren2]) THEN
  $FLAG[M_Test_GrdstFahren2]=TRUE
  UP_Rueckzug( )
  RETURN
ENDIF
;ENDFOLD

;-------------------------------
; Place part position
;-------------------------------
TRIGGER WHEN DISTANCE=1 DELAY=-1 DO Schrittmerker_R1Place(10753,10754,FPlace_R1_L7_S2_AP,XPlace_R1_L7_S2_AP) PRIO=-1
;FOLD LIN Place_R1_L7_S2_AP Vel=0.2 m/s LPlace_R1_L7_S2_AP Tool[1]:Upper Gripper Base[1]:Rack1;%{PE}%R8.3.21,%MKUKATPBASIS,%CMOVE,%VLIN,%P 1:LIN, 2:Place_R1_L7_S2_AP, 3:, 5:0.2, 7:LPlace_R1_L7_S2_AP
$BWDSTART=FALSE
LDAT_ACT= LLPlace_R1_L7_S2_AP
FDAT_ACT= FPlace_R1_L7_S2_AP
BAS(#CP_PARAMS,0.2)
LIN XPlace_R1_L7_S2_AP
;ENDFOLD

;FOLD Test the way back home - part 2
CONTINUE
IF $FLAG[M_Test_GrdstFahren2] THEN
  $FLAG[M_Test_GrdstFahren2]=FALSE
  UP_Rueckzug( )
  RETURN
ENDIF
;ENDFOLD

;***************************************************
; Disable part lost detection
SetPartLostDetection(NO_PART)
;***************************************************

TRIGGER WHEN DISTANCE=1 DELAY=-1 DO Schrittmerker_R1Place(10754,10755,FPlace_R1_L7_S2_NP1,XPlace_R1_L7_S2_NP1) PRIO=-1
;FOLD LIN Place_R1_L7_S2_NP1 Vel=0.2 m/s LPlace_R1_L7_S2_NP1 Tool[1]:Upper Gripper Base[1]:Rack1;%{PE}%R8.3.21,%MKUKATPBASIS,%CMOVE,%VLIN,%P 1:LIN, 2:Place_R1_L7_S2_NP1, 3:C_DIS C_DIS, 5:0.2, 7:LPlace_R1_L7_S2_NP1
$BWDSTART=FALSE
LDAT_ACT= LLPlace_R1_L7_S2_NP1
FDAT_ACT= FPlace_R1_L7_S2_NP1
BAS(#CP_PARAMS,0.2)
LIN XPlace_R1_L7_S2_NP1
;ENDFOLD

;***************************************************
; Check for part present (empty gripper)
CheckPartPresent(EMPTY_GRIPPER)
;***************************************************
; set load data
SetLoadData( )
;***************************************************

TRIGGER WHEN DISTANCE=1 DELAY=-1 DO Schrittmerker_R1Place(10755,10756,FPlace_R1_L7_S2_NP2,XPlace_R1_L7_S2_NP2) PRIO=-1
;FOLD LIN Place_R1_L7_S2_NP2 Vel=0.5 m/s LPlace_R1_L7_S2_NP2 Tool[1]:Upper Gripper Base[1]:Rack1;%{PE}%R8.3.21,%MKUKATPBASIS,%CMOVE,%VLIN,%P 1:LIN, 2:Place_R1_L7_S2_NP2, 3:, 5:0.5, 7:LPlace_R1_L7_S2_NP2
$BWDSTART=FALSE
LDAT_ACT= LLPlace_R1_L7_S2_NP2
FDAT_ACT= FPlace_R1_L7_S2_NP2
BAS(#CP_PARAMS,0.5)
LIN XPlace_R1_L7_S2_NP2
;ENDFOLD
TRIGGER WHEN DISTANCE=1 DELAY=-1 DO Schrittmerker_R1Place(10756,10757,FPlace_R1_L7_S2_NP3,XPlace_R1_L7_S2_NP3) PRIO=-1
;FOLD PTP Place_R1_L7_S2_NP3 CONT Vel=33 % PPlace_R1_L7_S2_NP3 Tool[1]:Upper Gripper Base[1]:Rack1;%{PE}%R8.3.21,%MKUKATPBASIS,%CMOVE,%VPTP,%P 1:PTP, 2:Place_R1_L7_S2_NP3, 3:C_DIS, 5:33, 7:PPlace_R1_L7_S2_NP3
$BWDSTART=FALSE
PDAT_ACT= PPPlace_R1_L7_S2_NP3
FDAT_ACT= FPlace_R1_L7_S2_NP3
BAS(#PTP_PARAMS,33)
PTP XPlace_R1_L7_S2_NP3 C_DIS
;ENDFOLD
TRIGGER WHEN DISTANCE=1 DELAY=-1 DO Schrittmerker_R1Place(10757,10758,FPlace_R1_L7_S2_NP4,XPlace_R1_L7_S2_NP4) PRIO=-1
;FOLD PTP Place_R1_L7_S2_NP4 CONT Vel=33 % PPlace_R1_L7_S2_NP4 Tool[1]:Upper Gripper Base[1]:Rack1;%{PE}%R8.3.21,%MKUKATPBASIS,%CMOVE,%VPTP,%P 1:PTP, 2:Place_R1_L7_S2_NP4, 3:C_DIS, 5:33, 7:PPlace_R1_L7_S2_NP4
$BWDSTART=FALSE
PDAT_ACT= PPPlace_R1_L7_S2_NP4
FDAT_ACT= FPlace_R1_L7_S2_NP4
BAS(#PTP_PARAMS,33)
PTP XPlace_R1_L7_S2_NP4 C_DIS
;ENDFOLD
TRIGGER WHEN DISTANCE=1 DELAY=-1 DO Schrittmerker_R1Place(10758,10759,FPlace_R1_L7_S2_NP5,XPlace_R1_L7_S2_NP5) PRIO=-1
;FOLD PTP Place_R1_L7_S2_NP5 CONT Vel=33 % PPlace_R1_L7_S2_NP5 Tool[1]:Upper Gripper Base[1]:Rack1;%{PE}%R8.3.21,%MKUKATPBASIS,%CMOVE,%VPTP,%P 1:PTP, 2:Place_R1_L7_S2_NP5, 3:C_DIS, 5:33, 7:PPlace_R1_L7_S2_NP5
$BWDSTART=FALSE
PDAT_ACT= PPPlace_R1_L7_S2_NP5
FDAT_ACT= FPlace_R1_L7_S2_NP5
BAS(#PTP_PARAMS,33)
PTP XPlace_R1_L7_S2_NP5 C_DIS
;ENDFOLD
TRIGGER WHEN DISTANCE=1 DELAY=-1 DO Schrittmerker_R1Place(10759,10760,FPlace_R1_L7_S2_NP6,XPlace_R1_L7_S2_NP6) PRIO=-1
;FOLD PTP Place_R1_L7_S2_NP6 CONT Vel=33 % PPlace_R1_L7_S2_NP6 Tool[1]:Upper Gripper Base[1]:Rack1;%{PE}%R8.3.21,%MKUKATPBASIS,%CMOVE,%VPTP,%P 1:PTP, 2:Place_R1_L7_S2_NP6, 3:C_DIS, 5:33, 7:PPlace_R1_L7_S2_NP6
$BWDSTART=FALSE
PDAT_ACT= PPPlace_R1_L7_S2_NP6
FDAT_ACT= FPlace_R1_L7_S2_NP6
BAS(#PTP_PARAMS,33)
PTP XPlace_R1_L7_S2_NP6 C_DIS
;ENDFOLD
TRIGGER WHEN DISTANCE=1 DELAY=-1 DO Schrittmerker_R1Place(10760,10761,FPlace_R1_L7_S2_NP7,XPlace_R1_L7_S2_NP7) PRIO=-1
;FOLD PTP Place_R1_L7_S2_NP7 CONT Vel=100 % PPlace_R1_L7_S2_NP7 Tool[1]:Upper Gripper Base[1]:Rack1;%{PE}%R8.3.21,%MKUKATPBASIS,%CMOVE,%VPTP,%P 1:PTP, 2:Place_R1_L7_S2_NP7, 3:C_DIS, 5:100, 7:PPlace_R1_L7_S2_NP7
$BWDSTART=FALSE
PDAT_ACT= PPPlace_R1_L7_S2_NP7
FDAT_ACT= FPlace_R1_L7_S2_NP7
BAS(#PTP_PARAMS,100)
PTP XPlace_R1_L7_S2_NP7 C_DIS
;ENDFOLD
TRIGGER WHEN DISTANCE=1 DELAY=-1 DO Schrittmerker_R1Place(10761,10762,FPlace_R1_L7_S2_NP8,XPlace_R1_L7_S2_NP8) PRIO=-1
;FOLD PTP Place_R1_L7_S2_NP8 CONT Vel=100 % PPlace_R1_L7_S2_NP8 Tool[1]:Upper Gripper Base[0];%{PE}%R8.3.21,%MKUKATPBASIS,%CMOVE,%VPTP,%P 1:PTP, 2:Place_R1_L7_S2_NP8, 3:C_DIS, 5:100, 7:PPlace_R1_L7_S2_NP8
$BWDSTART=FALSE
PDAT_ACT= PPPlace_R1_L7_S2_NP8
FDAT_ACT= FPlace_R1_L7_S2_NP8
BAS(#PTP_PARAMS,100)
PTP XPlace_R1_L7_S2_NP8 C_DIS
;ENDFOLD
TRIGGER WHEN DISTANCE=1 DELAY=-1 DO Schrittmerker_R1Place(10762,10763,FPlace_R1_L7_S2_NP9,XPlace_R1_L7_S2_NP9) PRIO=-1
;FOLD PTP Place_R1_L7_S2_NP9 CONT Vel=100 % PPlace_R1_L7_S2_NP9 Tool[1]:Upper Gripper Base[0];%{PE}%R8.3.21,%MKUKATPBASIS,%CMOVE,%VPTP,%P 1:PTP, 2:Place_R1_L7_S2_NP9, 3:C_DIS, 5:100, 7:PPlace_R1_L7_S2_NP9
$BWDSTART=FALSE
PDAT_ACT= PPPlace_R1_L7_S2_NP9
FDAT_ACT= FPlace_R1_L7_S2_NP9
BAS(#PTP_PARAMS,100)
PTP XPlace_R1_L7_S2_NP9 C_DIS
;ENDFOLD
TRIGGER WHEN DISTANCE=1 DELAY=-1 DO Schrittmerker_R1Place(10763,10764,FPlace_R1_L7_S2_NP10,XPlace_R1_L7_S2_NP10) PRIO=-1
;FOLD PTP Place_R1_L7_S2_NP10 CONT Vel=100 % PPlace_R1_L7_S2_NP10 Tool[1]:Upper Gripper Base[0];%{PE}%R8.3.21,%MKUKATPBASIS,%CMOVE,%VPTP,%P 1:PTP, 2:Place_R1_L7_S2_NP10, 3:C_DIS, 5:100, 7:PPlace_R1_L7_S2_NP10
$BWDSTART=FALSE
PDAT_ACT= PPPlace_R1_L7_S2_NP10
FDAT_ACT= FPlace_R1_L7_S2_NP10
BAS(#PTP_PARAMS,100)
PTP XPlace_R1_L7_S2_NP10 C_DIS
;ENDFOLD
TRIGGER WHEN DISTANCE=1 DELAY=-1 DO Schrittmerker_R1Place(10764,10765,FPlace_R1_L7_S2_NP11,XPlace_R1_L7_S2_NP11) PRIO=-1
;FOLD PTP Place_R1_L7_S2_NP11 CONT Vel=100 % PPlace_R1_L7_S2_NP11 Tool[1]:Upper Gripper Base[0];%{PE}%R8.3.21,%MKUKATPBASIS,%CMOVE,%VPTP,%P 1:PTP, 2:Place_R1_L7_S2_NP11, 3:C_DIS, 5:100, 7:PPlace_R1_L7_S2_NP11
$BWDSTART=FALSE
PDAT_ACT= PPPlace_R1_L7_S2_NP11
FDAT_ACT= FPlace_R1_L7_S2_NP11
BAS(#PTP_PARAMS,100)
PTP XPlace_R1_L7_S2_NP11 C_DIS
;ENDFOLD

TRIGGER WHEN DISTANCE=1 DELAY=-1 DO Schrittmerker_R1Place(10765,10501,FHOME,$nullframe,XHOME) PRIO=-1
;FOLD PTP HOME Vel=100 % PHome;%{PE}%R8.3.21,%MKUKATPBASIS,%CMOVE,%VPTP,%P 1:PTP, 2:HOME, 3:, 5:100, 7:PHome
$BWDSTART=FALSE
PDAT_ACT= PPHome
FDAT_ACT= FHOME
BAS(#PTP_PARAMS,100)
PTP XHOME
;ENDFOLD

;***************************************************
;FOLD Final tasks.
; Robot out of area Rack 1 Level 7
RobAusStorage1_7_A73=RESET_IN_AREA
;***************************************************
; stop cyclic clearence check
$CYCFLAG[ciFreigabeSPS]=DISABLE_MONITORING
;***************************************************
; Disable collision detection
;FOLD COLLDETECT Off ;%{PE}
;FOLD Parameters ;%{h}
;Params IlfProvider=kukaroboter.basistech.inlineforms.colldetect.off; CollDetect.Command=Off
;ENDFOLD
USE_CD_PARAMS(0)
;ENDFOLD
;***************************************************
;ENDFOLD
;***************************************************

END

; ##################################################

GLOBAL DEF UP_Place_R1_L7_S3( )
;***************************************************
; Place part on:
;    Rack  1
;    Level 7
;    Shelf 3
;***************************************************
;FOLD Preconditions - Vorraussetzungen
;***************************************************
; Enable collision detection
;FOLD COLLDETECT SetLimits Axis1: 150 % Axis2: 200 % Axis3: 150 % Axis4: 200 % Axis5: 150 % Axis6: 150 % ;%{PE}
;FOLD Parameters ;%{h}
;Params IlfProvider=kukaroboter.basistech.inlineforms.colldetect.setlimits; CollDetect.Command=SetLimits; CollDetect.Axis1=150; CollDetect.Axis2=200; CollDetect.Axis3=150; CollDetect.Axis4=200; CollDetect.Axis5=150; CollDetect.Axis6=150
;ENDFOLD
SET_TQ_VALUES(150, 200, 150, 200, 150, 150)
;ENDFOLD
;***************************************************
; Check for part in gripper (tool 1).
CheckPartPresent(OCCUPIED_GRIPPER,PART_ON_TOOL_1)
;***************************************************
; Enable part lost detection for tool 1
SetPartLostDetection(PART_ON_TOOL_1)
;***************************************************
; Set load data.
SetLoadData( )
;***************************************************
; Robot has to start from home position.
IF NOT $IN_HOME THEN
  UP_HomeToHome(0)
ENDIF
;***************************************************
;ENDFOLD

TRIGGER WHEN DISTANCE=1 DELAY=-1 DO Schrittmerker_R1Place(10501,10501,FHOME,$nullframe,XHOME) PRIO=-1
;FOLD PTP HOME Vel=12 % PHome;%{PE}%R8.3.21,%MKUKATPBASIS,%CMOVE,%VPTP,%P 1:PTP, 2:HOME, 3:, 5:12, 7:PHome
$BWDSTART=FALSE
PDAT_ACT= PPHome
FDAT_ACT= FHOME
BAS(#PTP_PARAMS,12)
PTP XHOME
;ENDFOLD

;***************************************************
;FOLD Area clearence handshake.
IF NOT $FLAG[M_Inbetriebnahme] THEN
  ;-------------------------------------------------
  ; Request area clearence.
  AnfStoer_Store1_7_A105=SET_REQUEST
  ;-------------------------------------------------
  ; Wait for area clearence from PLC.
  WAIT_FOR_INPUT("Frg_Storage1_7_E73",TRUE)
  ;-------------------------------------------------
  ; Reset area clearence request.
  AnfStoer_Store1_7_A105=RESET_REQUEST
  ;-------------------------------------------------
  ; start cyclic clearence check
  $CYCFLAG[ciFreigabeSPS]=Frg_Storage1_7_E73
  ;-------------------------------------------------
ENDIF
;***************************************************
; set "robot in area"
RobAusStorage1_7_A73=SET_IN_AREA
;ENDFOLD
;***************************************************

;***************************************************
;FOLD Check for Teachmode
IF $FLAG[M_Teachen] THEN
  WAIT FOR $T1
ENDIF
;ENDFOLD
;***************************************************

; move to the rack
TRIGGER WHEN DISTANCE=1 DELAY=-1 DO Schrittmerker_R1Place(10770,10501,FPlace_R1_L7_S3_VP1,XPlace_R1_L7_S3_VP1) PRIO=-1
;FOLD PTP Place_R1_L7_S3_VP1 CONT Vel=12 % PPlace_R1_L7_S3_VP1 Tool[1]:Upper Gripper Base[0];%{PE}%R8.3.21,%MKUKATPBASIS,%CMOVE,%VPTP,%P 1:PTP, 2:Place_R1_L7_S3_VP1, 3:C_DIS, 5:12, 7:PPlace_R1_L7_S3_VP1
$BWDSTART=FALSE
PDAT_ACT= PPPlace_R1_L7_S3_VP1
FDAT_ACT= FPlace_R1_L7_S3_VP1
BAS(#PTP_PARAMS,12)
PTP XPlace_R1_L7_S3_VP1 C_DIS
;ENDFOLD
TRIGGER WHEN DISTANCE=1 DELAY=-1 DO Schrittmerker_R1Place(10771,10770,FPlace_R1_L7_S3_VP2,XPlace_R1_L7_S3_VP2) PRIO=-1
;FOLD PTP Place_R1_L7_S3_VP2 CONT Vel=12 % PPlace_R1_L7_S3_VP2 Tool[1]:Upper Gripper Base[0];%{PE}%R8.3.21,%MKUKATPBASIS,%CMOVE,%VPTP,%P 1:PTP, 2:Place_R1_L7_S3_VP2, 3:C_DIS, 5:12, 7:PPlace_R1_L7_S3_VP2
$BWDSTART=FALSE
PDAT_ACT= PPPlace_R1_L7_S3_VP2
FDAT_ACT= FPlace_R1_L7_S3_VP2
BAS(#PTP_PARAMS,12)
PTP XPlace_R1_L7_S3_VP2 C_DIS
;ENDFOLD
TRIGGER WHEN DISTANCE=1 DELAY=-1 DO Schrittmerker_R1Place(10772,10771,FPlace_R1_L7_S3_VP3,XPlace_R1_L7_S3_VP3) PRIO=-1
;FOLD PTP Place_R1_L7_S3_VP3 CONT Vel=12 % PPlace_R1_L7_S3_VP3 Tool[1]:Upper Gripper Base[0];%{PE}%R8.3.21,%MKUKATPBASIS,%CMOVE,%VPTP,%P 1:PTP, 2:Place_R1_L7_S3_VP3, 3:C_DIS, 5:12, 7:PPlace_R1_L7_S3_VP3
$BWDSTART=FALSE
PDAT_ACT= PPPlace_R1_L7_S3_VP3
FDAT_ACT= FPlace_R1_L7_S3_VP3
BAS(#PTP_PARAMS,12)
PTP XPlace_R1_L7_S3_VP3 C_DIS
;ENDFOLD
TRIGGER WHEN DISTANCE=1 DELAY=-1 DO Schrittmerker_R1Place(10773,10772,FPlace_R1_L7_S3_VP4,XPlace_R1_L7_S3_VP4) PRIO=-1
;FOLD PTP Place_R1_L7_S3_VP4 CONT Vel=12 % PPlace_R1_L7_S3_VP4 Tool[1]:Upper Gripper Base[1]:Rack1;%{PE}%R8.3.21,%MKUKATPBASIS,%CMOVE,%VPTP,%P 1:PTP, 2:Place_R1_L7_S3_VP4, 3:C_DIS, 5:12, 7:PPlace_R1_L7_S3_VP4
$BWDSTART=FALSE
PDAT_ACT= PPPlace_R1_L7_S3_VP4
FDAT_ACT= FPlace_R1_L7_S3_VP4
BAS(#PTP_PARAMS,12)
PTP XPlace_R1_L7_S3_VP4 C_DIS
;ENDFOLD

TRIGGER WHEN DISTANCE=1 DELAY=-1 DO Schrittmerker_R1Place(10774,10773,FPlace_R1_L7_S3_Check,XPlace_R1_L7_S3_Check) PRIO=-1
;FOLD PTP Place_R1_L7_S3_Check Vel=12 % PPlace_R1_L7_S3_Check Tool[1]:Upper Gripper Base[1]:Rack1;%{PE}%R8.3.21,%MKUKATPBASIS,%CMOVE,%VPTP,%P 1:PTP, 2:Place_R1_L7_S3_Check, 3:, 5:12, 7:PPlace_R1_L7_S3_Check
$BWDSTART=FALSE
PDAT_ACT= PPPlace_R1_L7_S3_Check
FDAT_ACT= FPlace_R1_L7_S3_Check
BAS(#PTP_PARAMS,12)
PTP XPlace_R1_L7_S3_Check
;ENDFOLD

;***************************************************
;FOLD Pruefe Platz frei
IF (DetectPart(CHECK_SHELF,PLACE)==OCCUPIED) THEN
  UP_Rueckzug_R1Place( )
  RETURN
ENDIF
;ENDFOLD
;***************************************************

TRIGGER WHEN DISTANCE=1 DELAY=-1 DO Schrittmerker_R1Place(10775,10774,FPlace_R1_L7_S3_VP5,XPlace_R1_L7_S3_VP5) PRIO=-1
;FOLD LIN Place_R1_L7_S3_VP5 CONT Vel=0.5 m/s LPlace_R1_L7_S3_VP5 Tool[1]:Upper Gripper Base[1]:Rack1;%{PE}%R8.3.21,%MKUKATPBASIS,%CMOVE,%VLIN,%P 1:LIN, 2:Place_R1_L7_S3_VP5, 3:C_DIS C_DIS, 5:0.5, 7:LPlace_R1_L7_S3_VP5
$BWDSTART=FALSE
LDAT_ACT= LLPlace_R1_L7_S3_VP5
FDAT_ACT= FPlace_R1_L7_S3_VP5
BAS(#CP_PARAMS,0.5)
LIN XPlace_R1_L7_S3_VP5 C_DIS C_DIS
;ENDFOLD
TRIGGER WHEN DISTANCE=1 DELAY=-1 DO Schrittmerker_R1Place(10776,10775,FPlace_R1_L7_S3_VP6,XPlace_R1_L7_S3_VP6) PRIO=-1
;FOLD LIN Place_R1_L7_S3_VP6 CONT Vel=0.5 m/s LPlace_R1_L7_S3_VP6 Tool[1]:Upper Gripper Base[1]:Rack1;%{PE}%R8.3.21,%MKUKATPBASIS,%CMOVE,%VLIN,%P 1:LIN, 2:Place_R1_L7_S3_VP6, 3:C_DIS C_DIS, 5:0.5, 7:LPlace_R1_L7_S3_VP6
$BWDSTART=FALSE
LDAT_ACT= LLPlace_R1_L7_S3_VP6
FDAT_ACT= FPlace_R1_L7_S3_VP6
BAS(#CP_PARAMS,0.5)
LIN XPlace_R1_L7_S3_VP6 C_DIS C_DIS
;ENDFOLD
TRIGGER WHEN DISTANCE=1 DELAY=-1 DO Schrittmerker_R1Place(10777,10776,FPlace_R1_L7_S3_VP7,XPlace_R1_L7_S3_VP7) PRIO=-1
;FOLD LIN Place_R1_L7_S3_VP7 CONT Vel=0.5 m/s LPlace_R1_L7_S3_VP7 Tool[1]:Upper Gripper Base[1]:Rack1;%{PE}%R8.3.21,%MKUKATPBASIS,%CMOVE,%VLIN,%P 1:LIN, 2:Place_R1_L7_S3_VP7, 3:C_DIS C_DIS, 5:0.5, 7:LPlace_R1_L7_S3_VP7
$BWDSTART=FALSE
LDAT_ACT= LLPlace_R1_L7_S3_VP7
FDAT_ACT= FPlace_R1_L7_S3_VP7
BAS(#CP_PARAMS,0.5)
LIN XPlace_R1_L7_S3_VP7 C_DIS C_DIS
;ENDFOLD
TRIGGER WHEN DISTANCE=1 DELAY=-1 DO Schrittmerker_R1Place(10778,10777,FPlace_R1_L7_S3_VP8,XPlace_R1_L7_S3_VP8) PRIO=-1
;FOLD LIN Place_R1_L7_S3_VP8 CONT Vel=0.5 m/s LPlace_R1_L7_S3_VP8 Tool[1]:Upper Gripper Base[1]:Rack1;%{PE}%R8.3.21,%MKUKATPBASIS,%CMOVE,%VLIN,%P 1:LIN, 2:Place_R1_L7_S3_VP8, 3:C_DIS C_DIS, 5:0.5, 7:LPlace_R1_L7_S3_VP8
$BWDSTART=FALSE
LDAT_ACT= LLPlace_R1_L7_S3_VP8
FDAT_ACT= FPlace_R1_L7_S3_VP8
BAS(#CP_PARAMS,0.5)
LIN XPlace_R1_L7_S3_VP8 C_DIS C_DIS
;ENDFOLD

;FOLD Test the way back home - part 1
CONTINUE
IF ($FLAG[M_Test_GrdstFahren1] AND NOT $FLAG[M_Test_GrdstFahren2]) THEN
  $FLAG[M_Test_GrdstFahren2]=TRUE
  UP_Rueckzug( )
  RETURN
ENDIF
;ENDFOLD

;-------------------------------
; Place part position
;-------------------------------
TRIGGER WHEN DISTANCE=1 DELAY=-1 DO Schrittmerker_R1Place(10779,10780,FPlace_R1_L7_S3_AP,XPlace_R1_L7_S3_AP) PRIO=-1
;FOLD LIN Place_R1_L7_S3_AP Vel=0.2 m/s LPlace_R1_L7_S3_AP Tool[1]:Upper Gripper Base[1]:Rack1;%{PE}%R8.3.21,%MKUKATPBASIS,%CMOVE,%VLIN,%P 1:LIN, 2:Place_R1_L7_S3_AP, 3:, 5:0.2, 7:LPlace_R1_L7_S3_AP
$BWDSTART=FALSE
LDAT_ACT= LLPlace_R1_L7_S3_AP
FDAT_ACT= FPlace_R1_L7_S3_AP
BAS(#CP_PARAMS,0.2)
LIN XPlace_R1_L7_S3_AP
;ENDFOLD

;FOLD Test the way back home - part 2
CONTINUE
IF $FLAG[M_Test_GrdstFahren2] THEN
  $FLAG[M_Test_GrdstFahren2]=FALSE
  UP_Rueckzug( )
  RETURN
ENDIF
;ENDFOLD

;***************************************************
; Disable part lost detection
SetPartLostDetection(NO_PART)
;***************************************************

TRIGGER WHEN DISTANCE=1 DELAY=-1 DO Schrittmerker_R1Place(10780,10781,FPlace_R1_L7_S3_NP1,XPlace_R1_L7_S3_NP1) PRIO=-1
;FOLD LIN Place_R1_L7_S3_NP1 Vel=0.2 m/s LPlace_R1_L7_S3_NP1 Tool[1]:Upper Gripper Base[1]:Rack1;%{PE}%R8.3.21,%MKUKATPBASIS,%CMOVE,%VLIN,%P 1:LIN, 2:Place_R1_L7_S3_NP1, 3:C_DIS C_DIS, 5:0.2, 7:LPlace_R1_L7_S3_NP1
$BWDSTART=FALSE
LDAT_ACT= LLPlace_R1_L7_S3_NP1
FDAT_ACT= FPlace_R1_L7_S3_NP1
BAS(#CP_PARAMS,0.2)
LIN XPlace_R1_L7_S3_NP1
;ENDFOLD

;***************************************************
; Check for part present (empty gripper)
CheckPartPresent(EMPTY_GRIPPER)
;***************************************************
; set load data
SetLoadData( )
;***************************************************

TRIGGER WHEN DISTANCE=1 DELAY=-1 DO Schrittmerker_R1Place(10781,10782,FPlace_R1_L7_S3_NP2,XPlace_R1_L7_S3_NP2) PRIO=-1
;FOLD LIN Place_R1_L7_S3_NP2 Vel=0.5 m/s LPlace_R1_L7_S3_NP2 Tool[1]:Upper Gripper Base[1]:Rack1;%{PE}%R8.3.21,%MKUKATPBASIS,%CMOVE,%VLIN,%P 1:LIN, 2:Place_R1_L7_S3_NP2, 3:, 5:0.5, 7:LPlace_R1_L7_S3_NP2
$BWDSTART=FALSE
LDAT_ACT= LLPlace_R1_L7_S3_NP2
FDAT_ACT= FPlace_R1_L7_S3_NP2
BAS(#CP_PARAMS,0.5)
LIN XPlace_R1_L7_S3_NP2
;ENDFOLD
TRIGGER WHEN DISTANCE=1 DELAY=-1 DO Schrittmerker_R1Place(10782,10783,FPlace_R1_L7_S3_NP3,XPlace_R1_L7_S3_NP3) PRIO=-1
;FOLD PTP Place_R1_L7_S3_NP3 CONT Vel=33 % PPlace_R1_L7_S3_NP3 Tool[1]:Upper Gripper Base[1]:Rack1;%{PE}%R8.3.21,%MKUKATPBASIS,%CMOVE,%VPTP,%P 1:PTP, 2:Place_R1_L7_S3_NP3, 3:C_DIS, 5:33, 7:PPlace_R1_L7_S3_NP3
$BWDSTART=FALSE
PDAT_ACT= PPPlace_R1_L7_S3_NP3
FDAT_ACT= FPlace_R1_L7_S3_NP3
BAS(#PTP_PARAMS,33)
PTP XPlace_R1_L7_S3_NP3 C_DIS
;ENDFOLD
TRIGGER WHEN DISTANCE=1 DELAY=-1 DO Schrittmerker_R1Place(10783,10784,FPlace_R1_L7_S3_NP4,XPlace_R1_L7_S3_NP4) PRIO=-1
;FOLD PTP Place_R1_L7_S3_NP4 CONT Vel=33 % PPlace_R1_L7_S3_NP4 Tool[1]:Upper Gripper Base[1]:Rack1;%{PE}%R8.3.21,%MKUKATPBASIS,%CMOVE,%VPTP,%P 1:PTP, 2:Place_R1_L7_S3_NP4, 3:C_DIS, 5:33, 7:PPlace_R1_L7_S3_NP4
$BWDSTART=FALSE
PDAT_ACT= PPPlace_R1_L7_S3_NP4
FDAT_ACT= FPlace_R1_L7_S3_NP4
BAS(#PTP_PARAMS,33)
PTP XPlace_R1_L7_S3_NP4 C_DIS
;ENDFOLD
TRIGGER WHEN DISTANCE=1 DELAY=-1 DO Schrittmerker_R1Place(10784,10785,FPlace_R1_L7_S3_NP5,XPlace_R1_L7_S3_NP5) PRIO=-1
;FOLD PTP Place_R1_L7_S3_NP5 CONT Vel=33 % PPlace_R1_L7_S3_NP5 Tool[1]:Upper Gripper Base[1]:Rack1;%{PE}%R8.3.21,%MKUKATPBASIS,%CMOVE,%VPTP,%P 1:PTP, 2:Place_R1_L7_S3_NP5, 3:C_DIS, 5:33, 7:PPlace_R1_L7_S3_NP5
$BWDSTART=FALSE
PDAT_ACT= PPPlace_R1_L7_S3_NP5
FDAT_ACT= FPlace_R1_L7_S3_NP5
BAS(#PTP_PARAMS,33)
PTP XPlace_R1_L7_S3_NP5 C_DIS
;ENDFOLD
TRIGGER WHEN DISTANCE=1 DELAY=-1 DO Schrittmerker_R1Place(10785,10786,FPlace_R1_L7_S3_NP6,XPlace_R1_L7_S3_NP6) PRIO=-1
;FOLD PTP Place_R1_L7_S3_NP6 CONT Vel=100 % PPlace_R1_L7_S3_NP6 Tool[1]:Upper Gripper Base[0];%{PE}%R8.3.21,%MKUKATPBASIS,%CMOVE,%VPTP,%P 1:PTP, 2:Place_R1_L7_S3_NP6, 3:C_DIS, 5:100, 7:PPlace_R1_L7_S3_NP6
$BWDSTART=FALSE
PDAT_ACT= PPPlace_R1_L7_S3_NP6
FDAT_ACT= FPlace_R1_L7_S3_NP6
BAS(#PTP_PARAMS,100)
PTP XPlace_R1_L7_S3_NP6 C_DIS
;ENDFOLD
TRIGGER WHEN DISTANCE=1 DELAY=-1 DO Schrittmerker_R1Place(10786,10787,FPlace_R1_L7_S3_NP7,XPlace_R1_L7_S3_NP7) PRIO=-1
;FOLD PTP Place_R1_L7_S3_NP7 CONT Vel=100 % PPlace_R1_L7_S3_NP7 Tool[1]:Upper Gripper Base[0];%{PE}%R8.3.21,%MKUKATPBASIS,%CMOVE,%VPTP,%P 1:PTP, 2:Place_R1_L7_S3_NP7, 3:C_DIS, 5:100, 7:PPlace_R1_L7_S3_NP7
$BWDSTART=FALSE
PDAT_ACT= PPPlace_R1_L7_S3_NP7
FDAT_ACT= FPlace_R1_L7_S3_NP7
BAS(#PTP_PARAMS,100)
PTP XPlace_R1_L7_S3_NP7 C_DIS
;ENDFOLD
TRIGGER WHEN DISTANCE=1 DELAY=-1 DO Schrittmerker_R1Place(10787,10788,FPlace_R1_L7_S3_NP8,XPlace_R1_L7_S3_NP8) PRIO=-1
;FOLD PTP Place_R1_L7_S3_NP8 CONT Vel=100 % PPlace_R1_L7_S3_NP8 Tool[1]:Upper Gripper Base[0];%{PE}%R8.3.21,%MKUKATPBASIS,%CMOVE,%VPTP,%P 1:PTP, 2:Place_R1_L7_S3_NP8, 3:C_DIS, 5:100, 7:PPlace_R1_L7_S3_NP8
$BWDSTART=FALSE
PDAT_ACT= PPPlace_R1_L7_S3_NP8
FDAT_ACT= FPlace_R1_L7_S3_NP8
BAS(#PTP_PARAMS,100)
PTP XPlace_R1_L7_S3_NP8 C_DIS
;ENDFOLD

TRIGGER WHEN DISTANCE=1 DELAY=-1 DO Schrittmerker_R1Place(10788,10501,FHOME,$nullframe,XHOME) PRIO=-1
;FOLD PTP HOME Vel=100 % PHome;%{PE}%R8.3.21,%MKUKATPBASIS,%CMOVE,%VPTP,%P 1:PTP, 2:HOME, 3:, 5:100, 7:PHome
$BWDSTART=FALSE
PDAT_ACT= PPHome
FDAT_ACT= FHOME
BAS(#PTP_PARAMS,100)
PTP XHOME
;ENDFOLD

;***************************************************
;FOLD Final tasks.
; Robot out of area Rack 1 Level 7
RobAusStorage1_7_A73=RESET_IN_AREA
;***************************************************
; stop cyclic clearence check
$CYCFLAG[ciFreigabeSPS]=DISABLE_MONITORING
;***************************************************
; Disable collision detection
;FOLD COLLDETECT Off ;%{PE}
;FOLD Parameters ;%{h}
;Params IlfProvider=kukaroboter.basistech.inlineforms.colldetect.off; CollDetect.Command=Off
;ENDFOLD
USE_CD_PARAMS(0)
;ENDFOLD
;***************************************************
;ENDFOLD
;***************************************************

END

; ##################################################

GLOBAL DEF UP_Place_R1_L7_S4( )
;***************************************************
; Place part on:
;    Rack  1
;    Level 7
;    Shelf 4
;***************************************************
;FOLD Preconditions - Vorraussetzungen
;***************************************************
; Enable collision detection
;FOLD COLLDETECT SetLimits Axis1: 150 % Axis2: 200 % Axis3: 150 % Axis4: 200 % Axis5: 150 % Axis6: 150 % ;%{PE}
;FOLD Parameters ;%{h}
;Params IlfProvider=kukaroboter.basistech.inlineforms.colldetect.setlimits; CollDetect.Command=SetLimits; CollDetect.Axis1=150; CollDetect.Axis2=200; CollDetect.Axis3=150; CollDetect.Axis4=200; CollDetect.Axis5=150; CollDetect.Axis6=150
;ENDFOLD
SET_TQ_VALUES(150, 200, 150, 200, 150, 150)
;ENDFOLD
;***************************************************
; Check for part in gripper (tool 1).
CheckPartPresent(OCCUPIED_GRIPPER,PART_ON_TOOL_1)
;***************************************************
; Enable part lost detection for tool 1
SetPartLostDetection(PART_ON_TOOL_1)
;***************************************************
; Set load data.
SetLoadData( )
;***************************************************
; Robot has to start from home position.
IF NOT $IN_HOME THEN
  UP_HomeToHome(0)
ENDIF
;***************************************************
;ENDFOLD

TRIGGER WHEN DISTANCE=1 DELAY=-1 DO Schrittmerker_R1Place(10501,10501,FHOME,$nullframe,XHOME) PRIO=-1
;FOLD PTP HOME Vel=12 % PHome;%{PE}%R8.3.21,%MKUKATPBASIS,%CMOVE,%VPTP,%P 1:PTP, 2:HOME, 3:, 5:12, 7:PHome
$BWDSTART=FALSE
PDAT_ACT= PPHome
FDAT_ACT= FHOME
BAS(#PTP_PARAMS,12)
PTP XHOME
;ENDFOLD

;***************************************************
;FOLD Area clearence handshake.
IF NOT $FLAG[M_Inbetriebnahme] THEN
  ;-------------------------------------------------
  ; Request area clearence.
  AnfStoer_Store1_7_A105=SET_REQUEST
  ;-------------------------------------------------
  ; Wait for area clearence from PLC.
  WAIT_FOR_INPUT("Frg_Storage1_7_E73",TRUE)
  ;-------------------------------------------------
  ; Reset area clearence request.
  AnfStoer_Store1_7_A105=RESET_REQUEST
  ;-------------------------------------------------
  ; start cyclic clearence check
  $CYCFLAG[ciFreigabeSPS]=Frg_Storage1_7_E73
  ;-------------------------------------------------
ENDIF
;***************************************************
; set "robot in area"
RobAusStorage1_7_A73=SET_IN_AREA
;ENDFOLD
;***************************************************

;***************************************************
;FOLD Check for Teachmode
IF $FLAG[M_Teachen] THEN
  WAIT FOR $T1
ENDIF
;ENDFOLD
;***************************************************

; move to the rack
TRIGGER WHEN DISTANCE=1 DELAY=-1 DO Schrittmerker_R1Place(10800,10501,FPlace_R1_L7_S4_VP1,XPlace_R1_L7_S4_VP1) PRIO=-1
;FOLD PTP Place_R1_L7_S4_VP1 CONT Vel=12 % PPlace_R1_L7_S4_VP1 Tool[1]:Upper Gripper Base[0];%{PE}%R8.3.21,%MKUKATPBASIS,%CMOVE,%VPTP,%P 1:PTP, 2:Place_R1_L7_S4_VP1, 3:C_DIS, 5:12, 7:PPlace_R1_L7_S4_VP1
$BWDSTART=FALSE
PDAT_ACT= PPPlace_R1_L7_S4_VP1
FDAT_ACT= FPlace_R1_L7_S4_VP1
BAS(#PTP_PARAMS,12)
PTP XPlace_R1_L7_S4_VP1 C_DIS
;ENDFOLD
TRIGGER WHEN DISTANCE=1 DELAY=-1 DO Schrittmerker_R1Place(10801,10800,FPlace_R1_L7_S4_VP2,XPlace_R1_L7_S4_VP2) PRIO=-1
;FOLD PTP Place_R1_L7_S4_VP2 CONT Vel=12 % PPlace_R1_L7_S4_VP2 Tool[1]:Upper Gripper Base[0];%{PE}%R8.3.21,%MKUKATPBASIS,%CMOVE,%VPTP,%P 1:PTP, 2:Place_R1_L7_S4_VP2, 3:C_DIS, 5:12, 7:PPlace_R1_L7_S4_VP2
$BWDSTART=FALSE
PDAT_ACT= PPPlace_R1_L7_S4_VP2
FDAT_ACT= FPlace_R1_L7_S4_VP2
BAS(#PTP_PARAMS,12)
PTP XPlace_R1_L7_S4_VP2 C_DIS
;ENDFOLD
TRIGGER WHEN DISTANCE=1 DELAY=-1 DO Schrittmerker_R1Place(10802,10801,FPlace_R1_L7_S4_VP3,XPlace_R1_L7_S4_VP3) PRIO=-1
;FOLD PTP Place_R1_L7_S4_VP3 CONT Vel=12 % PPlace_R1_L7_S4_VP3 Tool[1]:Upper Gripper Base[0];%{PE}%R8.3.21,%MKUKATPBASIS,%CMOVE,%VPTP,%P 1:PTP, 2:Place_R1_L7_S4_VP3, 3:C_DIS, 5:12, 7:PPlace_R1_L7_S4_VP3
$BWDSTART=FALSE
PDAT_ACT= PPPlace_R1_L7_S4_VP3
FDAT_ACT= FPlace_R1_L7_S4_VP3
BAS(#PTP_PARAMS,12)
PTP XPlace_R1_L7_S4_VP3 C_DIS
;ENDFOLD

TRIGGER WHEN DISTANCE=1 DELAY=-1 DO Schrittmerker_R1Place(10803,10802,FPlace_R1_L7_S4_Check,XPlace_R1_L7_S4_Check) PRIO=-1
;FOLD PTP Place_R1_L7_S4_Check Vel=12 % PPlace_R1_L7_S4_Check Tool[1]:Upper Gripper Base[1]:Rack1;%{PE}%R8.3.21,%MKUKATPBASIS,%CMOVE,%VPTP,%P 1:PTP, 2:Place_R1_L7_S4_Check, 3:, 5:12, 7:PPlace_R1_L7_S4_Check
$BWDSTART=FALSE
PDAT_ACT= PPPlace_R1_L7_S4_Check
FDAT_ACT= FPlace_R1_L7_S4_Check
BAS(#PTP_PARAMS,12)
PTP XPlace_R1_L7_S4_Check
;ENDFOLD

;***************************************************
;FOLD Pruefe Platz frei
IF (DetectPart(CHECK_SHELF,PLACE)==OCCUPIED) THEN
  UP_Rueckzug_R1Place( )
  RETURN
ENDIF
;ENDFOLD
;***************************************************

TRIGGER WHEN DISTANCE=1 DELAY=-1 DO Schrittmerker_R1Place(10804,10803,FPlace_R1_L7_S4_VP4,XPlace_R1_L7_S4_VP4) PRIO=-1
;FOLD LIN Place_R1_L7_S4_VP4 CONT Vel=0.5 m/s LPlace_R1_L7_S4_VP4 Tool[1]:Upper Gripper Base[1]:Rack1;%{PE}%R8.3.21,%MKUKATPBASIS,%CMOVE,%VLIN,%P 1:LIN, 2:Place_R1_L7_S4_VP4, 3:C_DIS C_DIS, 5:0.5, 7:LPlace_R1_L7_S4_VP4
$BWDSTART=FALSE
LDAT_ACT= LLPlace_R1_L7_S4_VP4
FDAT_ACT= FPlace_R1_L7_S4_VP4
BAS(#CP_PARAMS,0.5)
LIN XPlace_R1_L7_S4_VP4 C_DIS C_DIS
;ENDFOLD
TRIGGER WHEN DISTANCE=1 DELAY=-1 DO Schrittmerker_R1Place(10805,10804,FPlace_R1_L7_S4_VP5,XPlace_R1_L7_S4_VP5) PRIO=-1
;FOLD LIN Place_R1_L7_S4_VP5 CONT Vel=0.5 m/s LPlace_R1_L7_S4_VP5 Tool[1]:Upper Gripper Base[1]:Rack1;%{PE}%R8.3.21,%MKUKATPBASIS,%CMOVE,%VLIN,%P 1:LIN, 2:Place_R1_L7_S4_VP5, 3:C_DIS C_DIS, 5:0.5, 7:LPlace_R1_L7_S4_VP5
$BWDSTART=FALSE
LDAT_ACT= LLPlace_R1_L7_S4_VP5
FDAT_ACT= FPlace_R1_L7_S4_VP5
BAS(#CP_PARAMS,0.5)
LIN XPlace_R1_L7_S4_VP5 C_DIS C_DIS
;ENDFOLD
TRIGGER WHEN DISTANCE=1 DELAY=-1 DO Schrittmerker_R1Place(10806,10805,FPlace_R1_L7_S4_VP6,XPlace_R1_L7_S4_VP6) PRIO=-1
;FOLD LIN Place_R1_L7_S4_VP6 CONT Vel=0.5 m/s LPlace_R1_L7_S4_VP6 Tool[1]:Upper Gripper Base[1]:Rack1;%{PE}%R8.3.21,%MKUKATPBASIS,%CMOVE,%VLIN,%P 1:LIN, 2:Place_R1_L7_S4_VP6, 3:C_DIS C_DIS, 5:0.5, 7:LPlace_R1_L7_S4_VP6
$BWDSTART=FALSE
LDAT_ACT= LLPlace_R1_L7_S4_VP6
FDAT_ACT= FPlace_R1_L7_S4_VP6
BAS(#CP_PARAMS,0.5)
LIN XPlace_R1_L7_S4_VP6 C_DIS C_DIS
;ENDFOLD

;FOLD Test the way back home - part 1
CONTINUE
IF ($FLAG[M_Test_GrdstFahren1] AND NOT $FLAG[M_Test_GrdstFahren2]) THEN
  $FLAG[M_Test_GrdstFahren2]=TRUE
  UP_Rueckzug( )
  RETURN
ENDIF
;ENDFOLD

;-------------------------------
; Place part position
;-------------------------------
TRIGGER WHEN DISTANCE=1 DELAY=-1 DO Schrittmerker_R1Place(10807,10808,FPlace_R1_L7_S4_AP,XPlace_R1_L7_S4_AP) PRIO=-1
;FOLD LIN Place_R1_L7_S4_AP Vel=0.2 m/s LPlace_R1_L7_S4_AP Tool[1]:Upper Gripper Base[1]:Rack1;%{PE}%R8.3.21,%MKUKATPBASIS,%CMOVE,%VLIN,%P 1:LIN, 2:Place_R1_L7_S4_AP, 3:, 5:0.2, 7:LPlace_R1_L7_S4_AP
$BWDSTART=FALSE
LDAT_ACT= LLPlace_R1_L7_S4_AP
FDAT_ACT= FPlace_R1_L7_S4_AP
BAS(#CP_PARAMS,0.2)
LIN XPlace_R1_L7_S4_AP
;ENDFOLD

;FOLD Test the way back home - part 2
CONTINUE
IF $FLAG[M_Test_GrdstFahren2] THEN
  $FLAG[M_Test_GrdstFahren2]=FALSE
  UP_Rueckzug( )
  RETURN
ENDIF
;ENDFOLD

;***************************************************
; Disable part lost detection
SetPartLostDetection(NO_PART)
;***************************************************

TRIGGER WHEN DISTANCE=1 DELAY=-1 DO Schrittmerker_R1Place(10808,10809,FPlace_R1_L7_S4_NP1,XPlace_R1_L7_S4_NP1) PRIO=-1
;FOLD LIN Place_R1_L7_S4_NP1 Vel=0.2 m/s LPlace_R1_L7_S4_NP1 Tool[1]:Upper Gripper Base[1]:Rack1;%{PE}%R8.3.21,%MKUKATPBASIS,%CMOVE,%VLIN,%P 1:LIN, 2:Place_R1_L7_S4_NP1, 3:C_DIS C_DIS, 5:0.2, 7:LPlace_R1_L7_S4_NP1
$BWDSTART=FALSE
LDAT_ACT= LLPlace_R1_L7_S4_NP1
FDAT_ACT= FPlace_R1_L7_S4_NP1
BAS(#CP_PARAMS,0.2)
LIN XPlace_R1_L7_S4_NP1
;ENDFOLD

;***************************************************
; Check for part present (empty gripper)
CheckPartPresent(EMPTY_GRIPPER)
;***************************************************
; set load data
SetLoadData( )
;***************************************************

TRIGGER WHEN DISTANCE=1 DELAY=-1 DO Schrittmerker_R1Place(10809,10810,FPlace_R1_L7_S4_NP2,XPlace_R1_L7_S4_NP2) PRIO=-1
;FOLD LIN Place_R1_L7_S4_NP2 CONT Vel=0.5 m/s LPlace_R1_L7_S4_NP2 Tool[1]:Upper Gripper Base[1]:Rack1;%{PE}%R8.3.21,%MKUKATPBASIS,%CMOVE,%VLIN,%P 1:LIN, 2:Place_R1_L7_S4_NP2, 3:C_DIS C_DIS, 5:0.5, 7:LPlace_R1_L7_S4_NP2
$BWDSTART=FALSE
LDAT_ACT= LLPlace_R1_L7_S4_NP2
FDAT_ACT= FPlace_R1_L7_S4_NP2
BAS(#CP_PARAMS,0.5)
LIN XPlace_R1_L7_S4_NP2 C_DIS C_DIS
;ENDFOLD
TRIGGER WHEN DISTANCE=1 DELAY=-1 DO Schrittmerker_R1Place(10810,10811,FPlace_R1_L7_S4_NP3,XPlace_R1_L7_S4_NP3) PRIO=-1
;FOLD LIN Place_R1_L7_S4_NP3 Vel=0.5 m/s LPlace_R1_L7_S4_NP3 Tool[1]:Upper Gripper Base[1]:Rack1;%{PE}%R8.3.21,%MKUKATPBASIS,%CMOVE,%VLIN,%P 1:LIN, 2:Place_R1_L7_S4_NP3, 3:, 5:0.5, 7:LPlace_R1_L7_S4_NP3
$BWDSTART=FALSE
LDAT_ACT= LLPlace_R1_L7_S4_NP3
FDAT_ACT= FPlace_R1_L7_S4_NP3
BAS(#CP_PARAMS,0.5)
LIN XPlace_R1_L7_S4_NP3
;ENDFOLD
TRIGGER WHEN DISTANCE=1 DELAY=-1 DO Schrittmerker_R1Place(10811,10812,FPlace_R1_L7_S4_NP4,XPlace_R1_L7_S4_NP4) PRIO=-1
;FOLD PTP Place_R1_L7_S4_NP4 CONT Vel=100 % PPlace_R1_L7_S4_NP4 Tool[1]:Upper Gripper Base[0];%{PE}%R8.3.21,%MKUKATPBASIS,%CMOVE,%VPTP,%P 1:PTP, 2:Place_R1_L7_S4_NP4, 3:C_DIS, 5:100, 7:PPlace_R1_L7_S4_NP4
$BWDSTART=FALSE
PDAT_ACT= PPPlace_R1_L7_S4_NP4
FDAT_ACT= FPlace_R1_L7_S4_NP4
BAS(#PTP_PARAMS,100)
PTP XPlace_R1_L7_S4_NP4 C_DIS
;ENDFOLD
TRIGGER WHEN DISTANCE=1 DELAY=-1 DO Schrittmerker_R1Place(10812,10813,FPlace_R1_L7_S4_NP5,XPlace_R1_L7_S4_NP5) PRIO=-1
;FOLD PTP Place_R1_L7_S4_NP5 CONT Vel=100 % PPlace_R1_L7_S4_NP5 Tool[1]:Upper Gripper Base[0];%{PE}%R8.3.21,%MKUKATPBASIS,%CMOVE,%VPTP,%P 1:PTP, 2:Place_R1_L7_S4_NP5, 3:C_DIS, 5:100, 7:PPlace_R1_L7_S4_NP5
$BWDSTART=FALSE
PDAT_ACT= PPPlace_R1_L7_S4_NP5
FDAT_ACT= FPlace_R1_L7_S4_NP5
BAS(#PTP_PARAMS,100)
PTP XPlace_R1_L7_S4_NP5 C_DIS
;ENDFOLD
TRIGGER WHEN DISTANCE=1 DELAY=-1 DO Schrittmerker_R1Place(10813,10814,FPlace_R1_L7_S4_NP6,XPlace_R1_L7_S4_NP6) PRIO=-1
;FOLD PTP Place_R1_L7_S4_NP6 CONT Vel=100 % PPlace_R1_L7_S4_NP6 Tool[1]:Upper Gripper Base[0];%{PE}%R8.3.21,%MKUKATPBASIS,%CMOVE,%VPTP,%P 1:PTP, 2:Place_R1_L7_S4_NP6, 3:C_DIS, 5:100, 7:PPlace_R1_L7_S4_NP6
$BWDSTART=FALSE
PDAT_ACT= PPPlace_R1_L7_S4_NP6
FDAT_ACT= FPlace_R1_L7_S4_NP6
BAS(#PTP_PARAMS,100)
PTP XPlace_R1_L7_S4_NP6 C_DIS
;ENDFOLD

TRIGGER WHEN DISTANCE=1 DELAY=-1 DO Schrittmerker_R1Place(10814,10501,FHOME,$nullframe,XHOME) PRIO=-1
;FOLD PTP HOME Vel=100 % PHome;%{PE}%R8.3.21,%MKUKATPBASIS,%CMOVE,%VPTP,%P 1:PTP, 2:HOME, 3:, 5:100, 7:PHome
$BWDSTART=FALSE
PDAT_ACT= PPHome
FDAT_ACT= FHOME
BAS(#PTP_PARAMS,100)
PTP XHOME
;ENDFOLD

;***************************************************
;FOLD Final tasks.
; Robot out of area Rack 1 Level 7
RobAusStorage1_7_A73=RESET_IN_AREA
;***************************************************
; stop cyclic clearence check
$CYCFLAG[ciFreigabeSPS]=DISABLE_MONITORING
;***************************************************
; Disable collision detection
;FOLD COLLDETECT Off ;%{PE}
;FOLD Parameters ;%{h}
;Params IlfProvider=kukaroboter.basistech.inlineforms.colldetect.off; CollDetect.Command=Off
;ENDFOLD
USE_CD_PARAMS(0)
;ENDFOLD
;***************************************************
;ENDFOLD
;***************************************************

END

; ##################################################

GLOBAL DEF UP_Place_R1_L8_S1( )
;***************************************************
; Place part on:
;    Rack  1
;    Level 8
;    Shelf 1
;***************************************************
;FOLD Preconditions - Vorraussetzungen
;***************************************************
; Enable collision detection
;FOLD COLLDETECT SetLimits Axis1: 150 % Axis2: 200 % Axis3: 150 % Axis4: 200 % Axis5: 150 % Axis6: 150 % ;%{PE}
;FOLD Parameters ;%{h}
;Params IlfProvider=kukaroboter.basistech.inlineforms.colldetect.setlimits; CollDetect.Command=SetLimits; CollDetect.Axis1=150; CollDetect.Axis2=200; CollDetect.Axis3=150; CollDetect.Axis4=200; CollDetect.Axis5=150; CollDetect.Axis6=150
;ENDFOLD
SET_TQ_VALUES(150, 200, 150, 200, 150, 150)
;ENDFOLD
;***************************************************
; Check for part in gripper (tool 1).
CheckPartPresent(OCCUPIED_GRIPPER,PART_ON_TOOL_1)
;***************************************************
; Enable part lost detection for tool 1
SetPartLostDetection(PART_ON_TOOL_1)
;***************************************************
; Set load data.
SetLoadData( )
;***************************************************
; Robot has to start from home position.
IF NOT $IN_HOME THEN
  UP_HomeToHome(0)
ENDIF
;***************************************************
;ENDFOLD

TRIGGER WHEN DISTANCE=1 DELAY=-1 DO Schrittmerker_R1Place(10501,10501,FHOME,$nullframe,XHOME) PRIO=-1
;FOLD PTP HOME Vel=12 % PHome;%{PE}%R8.3.21,%MKUKATPBASIS,%CMOVE,%VPTP,%P 1:PTP, 2:HOME, 3:, 5:12, 7:PHome
$BWDSTART=FALSE
PDAT_ACT= PPHome
FDAT_ACT= FHOME
BAS(#PTP_PARAMS,12)
PTP XHOME
;ENDFOLD

;***************************************************
;FOLD Area clearence handshake.
IF NOT $FLAG[M_Inbetriebnahme] THEN
  ;-------------------------------------------------
  ; Request area clearence.
  AnfStoer_Store1_8_A106=SET_REQUEST
  ;-------------------------------------------------
  ; Wait for area clearence from PLC.
  WAIT_FOR_INPUT("Frg_Storage1_8_E74",TRUE)
  ;-------------------------------------------------
  ; Reset area clearence request.
  AnfStoer_Store1_8_A106=RESET_REQUEST
  ;-------------------------------------------------
  ; start cyclic clearence check
  $CYCFLAG[ciFreigabeSPS]=Frg_Storage1_8_E74
  ;-------------------------------------------------
ENDIF
;***************************************************
; set "robot in area"
RobAusStorage1_8_A74=SET_IN_AREA
;ENDFOLD
;***************************************************

;***************************************************
;FOLD Check for Teachmode
IF $FLAG[M_Teachen] THEN
  WAIT FOR $T1
ENDIF
;ENDFOLD
;***************************************************

; move to the rack
TRIGGER WHEN DISTANCE=1 DELAY=-1 DO Schrittmerker_R1Place(10820,10501,FPlace_R1_L8_S1_VP1,XPlace_R1_L8_S1_VP1) PRIO=-1
;FOLD PTP Place_R1_L8_S1_VP1 CONT Vel=12 % PPlace_R1_L8_S1_VP1 Tool[1]:Upper Gripper Base[0];%{PE}%R8.3.21,%MKUKATPBASIS,%CMOVE,%VPTP,%P 1:PTP, 2:Place_R1_L8_S1_VP1, 3:C_DIS, 5:12, 7:PPlace_R1_L8_S1_VP1
$BWDSTART=FALSE
PDAT_ACT= PPPlace_R1_L8_S1_VP1
FDAT_ACT= FPlace_R1_L8_S1_VP1
BAS(#PTP_PARAMS,12)
PTP XPlace_R1_L8_S1_VP1 C_DIS
;ENDFOLD
TRIGGER WHEN DISTANCE=1 DELAY=-1 DO Schrittmerker_R1Place(10821,10820,FPlace_R1_L8_S1_VP2,XPlace_R1_L8_S1_VP2) PRIO=-1
;FOLD PTP Place_R1_L8_S1_VP2 CONT Vel=12 % PPlace_R1_L8_S1_VP2 Tool[1]:Upper Gripper Base[0];%{PE}%R8.3.21,%MKUKATPBASIS,%CMOVE,%VPTP,%P 1:PTP, 2:Place_R1_L8_S1_VP2, 3:C_DIS, 5:12, 7:PPlace_R1_L8_S1_VP2
$BWDSTART=FALSE
PDAT_ACT= PPPlace_R1_L8_S1_VP2
FDAT_ACT= FPlace_R1_L8_S1_VP2
BAS(#PTP_PARAMS,12)
PTP XPlace_R1_L8_S1_VP2 C_DIS
;ENDFOLD
TRIGGER WHEN DISTANCE=1 DELAY=-1 DO Schrittmerker_R1Place(10822,10821,FPlace_R1_L8_S1_VP3,XPlace_R1_L8_S1_VP3) PRIO=-1
;FOLD PTP Place_R1_L8_S1_VP3 CONT Vel=12 % PPlace_R1_L8_S1_VP3 Tool[1]:Upper Gripper Base[0];%{PE}%R8.3.21,%MKUKATPBASIS,%CMOVE,%VPTP,%P 1:PTP, 2:Place_R1_L8_S1_VP3, 3:C_DIS, 5:12, 7:PPlace_R1_L8_S1_VP3
$BWDSTART=FALSE
PDAT_ACT= PPPlace_R1_L8_S1_VP3
FDAT_ACT= FPlace_R1_L8_S1_VP3
BAS(#PTP_PARAMS,12)
PTP XPlace_R1_L8_S1_VP3 C_DIS
;ENDFOLD
TRIGGER WHEN DISTANCE=1 DELAY=-1 DO Schrittmerker_R1Place(10823,10822,FPlace_R1_L8_S1_VP4,XPlace_R1_L8_S1_VP4) PRIO=-1
;FOLD PTP Place_R1_L8_S1_VP4 CONT Vel=12 % PPlace_R1_L8_S1_VP4 Tool[1]:Upper Gripper Base[0];%{PE}%R8.3.21,%MKUKATPBASIS,%CMOVE,%VPTP,%P 1:PTP, 2:Place_R1_L8_S1_VP4, 3:C_DIS, 5:12, 7:PPlace_R1_L8_S1_VP4
$BWDSTART=FALSE
PDAT_ACT= PPPlace_R1_L8_S1_VP4
FDAT_ACT= FPlace_R1_L8_S1_VP4
BAS(#PTP_PARAMS,12)
PTP XPlace_R1_L8_S1_VP4 C_DIS
;ENDFOLD
TRIGGER WHEN DISTANCE=1 DELAY=-1 DO Schrittmerker_R1Place(10824,10823,FPlace_R1_L8_S1_VP5,XPlace_R1_L8_S1_VP5) PRIO=-1
;FOLD PTP Place_R1_L8_S1_VP5 CONT Vel=12 % PPlace_R1_L8_S1_VP5 Tool[1]:Upper Gripper Base[0];%{PE}%R8.3.21,%MKUKATPBASIS,%CMOVE,%VPTP,%P 1:PTP, 2:Place_R1_L8_S1_VP5, 3:C_DIS, 5:12, 7:PPlace_R1_L8_S1_VP5
$BWDSTART=FALSE
PDAT_ACT= PPPlace_R1_L8_S1_VP5
FDAT_ACT= FPlace_R1_L8_S1_VP5
BAS(#PTP_PARAMS,12)
PTP XPlace_R1_L8_S1_VP5 C_DIS
;ENDFOLD
TRIGGER WHEN DISTANCE=1 DELAY=-1 DO Schrittmerker_R1Place(10825,10824,FPlace_R1_L8_S1_VP6,XPlace_R1_L8_S1_VP6) PRIO=-1
;FOLD PTP Place_R1_L8_S1_VP6 CONT Vel=12 % PPlace_R1_L8_S1_VP6 Tool[1]:Upper Gripper Base[1]:Rack1;%{PE}%R8.3.21,%MKUKATPBASIS,%CMOVE,%VPTP,%P 1:PTP, 2:Place_R1_L8_S1_VP6, 3:C_DIS, 5:12, 7:PPlace_R1_L8_S1_VP6
$BWDSTART=FALSE
PDAT_ACT= PPPlace_R1_L8_S1_VP6
FDAT_ACT= FPlace_R1_L8_S1_VP6
BAS(#PTP_PARAMS,12)
PTP XPlace_R1_L8_S1_VP6 C_DIS
;ENDFOLD
TRIGGER WHEN DISTANCE=1 DELAY=-1 DO Schrittmerker_R1Place(10826,10825,FPlace_R1_L8_S1_VP7,XPlace_R1_L8_S1_VP7) PRIO=-1
;FOLD PTP Place_R1_L8_S1_VP7 CONT Vel=12 % PPlace_R1_L8_S1_VP7 Tool[1]:Upper Gripper Base[1]:Rack1;%{PE}%R8.3.21,%MKUKATPBASIS,%CMOVE,%VPTP,%P 1:PTP, 2:Place_R1_L8_S1_VP7, 3:C_DIS, 5:12, 7:PPlace_R1_L8_S1_VP7
$BWDSTART=FALSE
PDAT_ACT= PPPlace_R1_L8_S1_VP7
FDAT_ACT= FPlace_R1_L8_S1_VP7
BAS(#PTP_PARAMS,12)
PTP XPlace_R1_L8_S1_VP7 C_DIS
;ENDFOLD
TRIGGER WHEN DISTANCE=1 DELAY=-1 DO Schrittmerker_R1Place(10827,10826,FPlace_R1_L8_S1_VP8,XPlace_R1_L8_S1_VP8) PRIO=-1
;FOLD PTP Place_R1_L8_S1_VP8 CONT Vel=12 % PPlace_R1_L8_S1_VP8 Tool[1]:Upper Gripper Base[1]:Rack1;%{PE}%R8.3.21,%MKUKATPBASIS,%CMOVE,%VPTP,%P 1:PTP, 2:Place_R1_L8_S1_VP8, 3:C_DIS, 5:12, 7:PPlace_R1_L8_S1_VP8
$BWDSTART=FALSE
PDAT_ACT= PPPlace_R1_L8_S1_VP8
FDAT_ACT= FPlace_R1_L8_S1_VP8
BAS(#PTP_PARAMS,12)
PTP XPlace_R1_L8_S1_VP8 C_DIS
;ENDFOLD

TRIGGER WHEN DISTANCE=1 DELAY=-1 DO Schrittmerker_R1Place(10828,10827,FPlace_R1_L8_S1_Check,XPlace_R1_L8_S1_Check) PRIO=-1
;FOLD PTP Place_R1_L8_S1_Check Vel=12 % PPlace_R1_L8_S1_Check Tool[1]:Upper Gripper Base[1]:Rack1;%{PE}%R8.3.21,%MKUKATPBASIS,%CMOVE,%VPTP,%P 1:PTP, 2:Place_R1_L8_S1_Check, 3:, 5:12, 7:PPlace_R1_L8_S1_Check
$BWDSTART=FALSE
PDAT_ACT= PPPlace_R1_L8_S1_Check
FDAT_ACT= FPlace_R1_L8_S1_Check
BAS(#PTP_PARAMS,12)
PTP XPlace_R1_L8_S1_Check
;ENDFOLD

;***************************************************
;FOLD Pruefe Platz frei
IF (DetectPart(CHECK_SHELF,PLACE)==OCCUPIED) THEN
  UP_Rueckzug_R1Place( )
  RETURN
ENDIF
;ENDFOLD
;***************************************************

TRIGGER WHEN DISTANCE=1 DELAY=-1 DO Schrittmerker_R1Place(10829,10828,FPlace_R1_L8_S1_VP9,XPlace_R1_L8_S1_VP9) PRIO=-1
;FOLD LIN Place_R1_L8_S1_VP9 CONT Vel=0.5 m/s LPlace_R1_L8_S1_VP9 Tool[1]:Upper Gripper Base[1]:Rack1;%{PE}%R8.3.21,%MKUKATPBASIS,%CMOVE,%VLIN,%P 1:LIN, 2:Place_R1_L8_S1_VP9, 3:C_DIS C_DIS, 5:0.5, 7:LPlace_R1_L8_S1_VP9
$BWDSTART=FALSE
LDAT_ACT= LLPlace_R1_L8_S1_VP9
FDAT_ACT= FPlace_R1_L8_S1_VP9
BAS(#CP_PARAMS,0.5)
LIN XPlace_R1_L8_S1_VP9 C_DIS C_DIS
;ENDFOLD

;***************************************************
;FOLD Test the way back home - part 1
CONTINUE
IF ($FLAG[M_Test_GrdstFahren1] AND NOT $FLAG[M_Test_GrdstFahren2]) THEN
  $FLAG[M_Test_GrdstFahren2]=TRUE
  UP_Rueckzug( )
  RETURN
ENDIF
;ENDFOLD
;***************************************************

;-------------------------------
; Place part position
;-------------------------------
TRIGGER WHEN DISTANCE=1 DELAY=-1 DO Schrittmerker_R1Place(10830,10831,FPlace_R1_L8_S1_AP,XPlace_R1_L8_S1_AP) PRIO=-1
;FOLD LIN Place_R1_L8_S1_AP Vel=0.2 m/s LPlace_R1_L8_S1_AP Tool[1]:Upper Gripper Base[1]:Rack1;%{PE}%R8.3.21,%MKUKATPBASIS,%CMOVE,%VLIN,%P 1:LIN, 2:Place_R1_L8_S1_AP, 3:, 5:0.2, 7:LPlace_R1_L8_S1_AP
$BWDSTART=FALSE
LDAT_ACT= LLPlace_R1_L8_S1_AP
FDAT_ACT= FPlace_R1_L8_S1_AP
BAS(#CP_PARAMS,0.2)
LIN XPlace_R1_L8_S1_AP
;ENDFOLD

;FOLD Test the way back home - part 2
CONTINUE
IF $FLAG[M_Test_GrdstFahren2] THEN
  $FLAG[M_Test_GrdstFahren2]=FALSE
  UP_Rueckzug( )
  RETURN
ENDIF
;ENDFOLD

;***************************************************
; Disable part lost detection
SetPartLostDetection(NO_PART)
;***************************************************

TRIGGER WHEN DISTANCE=1 DELAY=-1 DO Schrittmerker_R1Place(10831,10832,FPlace_R1_L8_S1_NP1,XPlace_R1_L8_S1_NP1) PRIO=-1
;FOLD LIN Place_R1_L8_S1_NP1 Vel=0.2 m/s LPlace_R1_L8_S1_NP1 Tool[1]:Upper Gripper Base[1]:Rack1;%{PE}%R8.3.21,%MKUKATPBASIS,%CMOVE,%VLIN,%P 1:LIN, 2:Place_R1_L8_S1_NP1, 3:C_DIS C_DIS, 5:0.2, 7:LPlace_R1_L8_S1_NP1
$BWDSTART=FALSE
LDAT_ACT= LLPlace_R1_L8_S1_NP1
FDAT_ACT= FPlace_R1_L8_S1_NP1
BAS(#CP_PARAMS,0.2)
LIN XPlace_R1_L8_S1_NP1
;ENDFOLD

;***************************************************
; Check for part present (empty gripper)
CheckPartPresent(EMPTY_GRIPPER)
;***************************************************
; set load data
SetLoadData( )
;***************************************************

TRIGGER WHEN DISTANCE=1 DELAY=-1 DO Schrittmerker_R1Place(10832,10833,FPlace_R1_L8_S1_NP2,XPlace_R1_L8_S1_NP2) PRIO=-1
;FOLD LIN Place_R1_L8_S1_NP2 Vel=0.5 m/s LPlace_R1_L8_S1_NP2 Tool[1]:Upper Gripper Base[1]:Rack1;%{PE}%R8.3.21,%MKUKATPBASIS,%CMOVE,%VLIN,%P 1:LIN, 2:Place_R1_L8_S1_NP2, 3:, 5:0.5, 7:LPlace_R1_L8_S1_NP2
$BWDSTART=FALSE
LDAT_ACT= LLPlace_R1_L8_S1_NP2
FDAT_ACT= FPlace_R1_L8_S1_NP2
BAS(#CP_PARAMS,0.5)
LIN XPlace_R1_L8_S1_NP2
;ENDFOLD
TRIGGER WHEN DISTANCE=1 DELAY=-1 DO Schrittmerker_R1Place(10833,10834,FPlace_R1_L8_S1_NP3,XPlace_R1_L8_S1_NP3) PRIO=-1
;FOLD PTP Place_R1_L8_S1_NP3 CONT Vel=100 % PPlace_R1_L8_S1_NP3 Tool[1]:Upper Gripper Base[0];%{PE}%R8.3.21,%MKUKATPBASIS,%CMOVE,%VPTP,%P 1:PTP, 2:Place_R1_L8_S1_NP3, 3:C_DIS, 5:100, 7:PPlace_R1_L8_S1_NP3
$BWDSTART=FALSE
PDAT_ACT= PPPlace_R1_L8_S1_NP3
FDAT_ACT= FPlace_R1_L8_S1_NP3
BAS(#PTP_PARAMS,100)
PTP XPlace_R1_L8_S1_NP3 C_DIS
;ENDFOLD
TRIGGER WHEN DISTANCE=1 DELAY=-1 DO Schrittmerker_R1Place(10834,10835,FPlace_R1_L8_S1_NP4,XPlace_R1_L8_S1_NP4) PRIO=-1
;FOLD PTP Place_R1_L8_S1_NP4 CONT Vel=100 % PPlace_R1_L8_S1_NP4 Tool[1]:Upper Gripper Base[0];%{PE}%R8.3.21,%MKUKATPBASIS,%CMOVE,%VPTP,%P 1:PTP, 2:Place_R1_L8_S1_NP4, 3:C_DIS, 5:100, 7:PPlace_R1_L8_S1_NP4
$BWDSTART=FALSE
PDAT_ACT= PPPlace_R1_L8_S1_NP4
FDAT_ACT= FPlace_R1_L8_S1_NP4
BAS(#PTP_PARAMS,100)
PTP XPlace_R1_L8_S1_NP4 C_DIS
;ENDFOLD

TRIGGER WHEN DISTANCE=1 DELAY=-1 DO Schrittmerker_R1Place(10835,10501,FHOME,$nullframe,XHOME) PRIO=-1
;FOLD PTP HOME Vel=100 % PHome;%{PE}%R8.3.21,%MKUKATPBASIS,%CMOVE,%VPTP,%P 1:PTP, 2:HOME, 3:, 5:100, 7:PHome
$BWDSTART=FALSE
PDAT_ACT= PPHome
FDAT_ACT= FHOME
BAS(#PTP_PARAMS,100)
PTP XHOME
;ENDFOLD

;***************************************************
;FOLD Final tasks.
; Robot out of area Rack 1 Level 8
RobAusStorage1_8_A74=RESET_IN_AREA
;***************************************************
; stop cyclic clearence check
$CYCFLAG[ciFreigabeSPS]=DISABLE_MONITORING
;***************************************************
; Disable collision detection
;FOLD COLLDETECT Off ;%{PE}
;FOLD Parameters ;%{h}
;Params IlfProvider=kukaroboter.basistech.inlineforms.colldetect.off; CollDetect.Command=Off
;ENDFOLD
USE_CD_PARAMS(0)
;ENDFOLD
;***************************************************
;ENDFOLD
;***************************************************

END

; ##################################################

GLOBAL DEF UP_Place_R1_L8_S2( )
;***************************************************
; Place part on:
;    Rack  1
;    Level 8
;    Shelf 2
;***************************************************
;FOLD Preconditions - Vorraussetzungen
;***************************************************
; Enable collision detection
;FOLD COLLDETECT SetLimits Axis1: 150 % Axis2: 200 % Axis3: 150 % Axis4: 200 % Axis5: 150 % Axis6: 150 % ;%{PE}
;FOLD Parameters ;%{h}
;Params IlfProvider=kukaroboter.basistech.inlineforms.colldetect.setlimits; CollDetect.Command=SetLimits; CollDetect.Axis1=150; CollDetect.Axis2=200; CollDetect.Axis3=150; CollDetect.Axis4=200; CollDetect.Axis5=150; CollDetect.Axis6=150
;ENDFOLD
SET_TQ_VALUES(150, 200, 150, 200, 150, 150)
;ENDFOLD
;***************************************************
; Check for part in gripper (tool 1).
CheckPartPresent(OCCUPIED_GRIPPER,PART_ON_TOOL_1)
;***************************************************
; Enable part lost detection for tool 1
SetPartLostDetection(PART_ON_TOOL_1)
;***************************************************
; Set load data.
SetLoadData( )
;***************************************************
; Robot has to start from home position.
IF NOT $IN_HOME THEN
  UP_HomeToHome(0)
ENDIF
;***************************************************
;ENDFOLD

TRIGGER WHEN DISTANCE=1 DELAY=-1 DO Schrittmerker_R1Place(10501,10501,FHOME,$nullframe,XHOME) PRIO=-1
;FOLD PTP HOME Vel=12 % PHome;%{PE}%R8.3.21,%MKUKATPBASIS,%CMOVE,%VPTP,%P 1:PTP, 2:HOME, 3:, 5:12, 7:PHome
$BWDSTART=FALSE
PDAT_ACT= PPHome
FDAT_ACT= FHOME
BAS(#PTP_PARAMS,12)
PTP XHOME
;ENDFOLD

;***************************************************
;FOLD Area clearence handshake.
IF NOT $FLAG[M_Inbetriebnahme] THEN
  ;-------------------------------------------------
  ; Request area clearence.
  AnfStoer_Store1_8_A106=SET_REQUEST
  ;-------------------------------------------------
  ; Wait for area clearence from PLC.
  WAIT_FOR_INPUT("Frg_Storage1_8_E74",TRUE)
  ;-------------------------------------------------
  ; Reset area clearence request.
  AnfStoer_Store1_8_A106=RESET_REQUEST
  ;-------------------------------------------------
  ; start cyclic clearence check
  $CYCFLAG[ciFreigabeSPS]=Frg_Storage1_8_E74
  ;-------------------------------------------------
ENDIF
;***************************************************
; set "robot in area"
RobAusStorage1_8_A74=SET_IN_AREA
;ENDFOLD
;***************************************************

;***************************************************
;FOLD Check for Teachmode
IF $FLAG[M_Teachen] THEN
  WAIT FOR $T1
ENDIF
;ENDFOLD
;***************************************************

; move to the rack
TRIGGER WHEN DISTANCE=1 DELAY=-1 DO Schrittmerker_R1Place(10840,10501,FPlace_R1_L8_S2_VP1,XPlace_R1_L8_S2_VP1) PRIO=-1
;FOLD PTP Place_R1_L8_S2_VP1 CONT Vel=12 % PPlace_R1_L8_S2_VP1 Tool[1]:Upper Gripper Base[0];%{PE}%R8.3.21,%MKUKATPBASIS,%CMOVE,%VPTP,%P 1:PTP, 2:Place_R1_L8_S2_VP1, 3:C_DIS, 5:12, 7:PPlace_R1_L8_S2_VP1
$BWDSTART=FALSE
PDAT_ACT= PPPlace_R1_L8_S2_VP1
FDAT_ACT= FPlace_R1_L8_S2_VP1
BAS(#PTP_PARAMS,12)
PTP XPlace_R1_L8_S2_VP1 C_DIS
;ENDFOLD
TRIGGER WHEN DISTANCE=1 DELAY=-1 DO Schrittmerker_R1Place(10841,10840,FPlace_R1_L8_S2_VP2,XPlace_R1_L8_S2_VP2) PRIO=-1
;FOLD PTP Place_R1_L8_S2_VP2 CONT Vel=12 % PPlace_R1_L8_S2_VP2 Tool[1]:Upper Gripper Base[0];%{PE}%R8.3.21,%MKUKATPBASIS,%CMOVE,%VPTP,%P 1:PTP, 2:Place_R1_L8_S2_VP2, 3:C_DIS, 5:12, 7:PPlace_R1_L8_S2_VP2
$BWDSTART=FALSE
PDAT_ACT= PPPlace_R1_L8_S2_VP2
FDAT_ACT= FPlace_R1_L8_S2_VP2
BAS(#PTP_PARAMS,12)
PTP XPlace_R1_L8_S2_VP2 C_DIS
;ENDFOLD
TRIGGER WHEN DISTANCE=1 DELAY=-1 DO Schrittmerker_R1Place(10842,10841,FPlace_R1_L8_S2_VP3,XPlace_R1_L8_S2_VP3) PRIO=-1
;FOLD PTP Place_R1_L8_S2_VP3 CONT Vel=12 % PPlace_R1_L8_S2_VP3 Tool[1]:Upper Gripper Base[0];%{PE}%R8.3.21,%MKUKATPBASIS,%CMOVE,%VPTP,%P 1:PTP, 2:Place_R1_L8_S2_VP3, 3:C_DIS, 5:12, 7:PPlace_R1_L8_S2_VP3
$BWDSTART=FALSE
PDAT_ACT= PPPlace_R1_L8_S2_VP3
FDAT_ACT= FPlace_R1_L8_S2_VP3
BAS(#PTP_PARAMS,12)
PTP XPlace_R1_L8_S2_VP3 C_DIS
;ENDFOLD
TRIGGER WHEN DISTANCE=1 DELAY=-1 DO Schrittmerker_R1Place(10843,10842,FPlace_R1_L8_S2_VP4,XPlace_R1_L8_S2_VP4) PRIO=-1
;FOLD PTP Place_R1_L8_S2_VP4 CONT Vel=12 % PPlace_R1_L8_S2_VP4 Tool[1]:Upper Gripper Base[0];%{PE}%R8.3.21,%MKUKATPBASIS,%CMOVE,%VPTP,%P 1:PTP, 2:Place_R1_L8_S2_VP4, 3:C_DIS, 5:12, 7:PPlace_R1_L8_S2_VP4
$BWDSTART=FALSE
PDAT_ACT= PPPlace_R1_L8_S2_VP4
FDAT_ACT= FPlace_R1_L8_S2_VP4
BAS(#PTP_PARAMS,12)
PTP XPlace_R1_L8_S2_VP4 C_DIS
;ENDFOLD
TRIGGER WHEN DISTANCE=1 DELAY=-1 DO Schrittmerker_R1Place(10844,10843,FPlace_R1_L8_S2_VP5,XPlace_R1_L8_S2_VP5) PRIO=-1
;FOLD PTP Place_R1_L8_S2_VP5 CONT Vel=12 % PPlace_R1_L8_S2_VP5 Tool[1]:Upper Gripper Base[0];%{PE}%R8.3.21,%MKUKATPBASIS,%CMOVE,%VPTP,%P 1:PTP, 2:Place_R1_L8_S2_VP5, 3:C_DIS, 5:12, 7:PPlace_R1_L8_S2_VP5
$BWDSTART=FALSE
PDAT_ACT= PPPlace_R1_L8_S2_VP5
FDAT_ACT= FPlace_R1_L8_S2_VP5
BAS(#PTP_PARAMS,12)
PTP XPlace_R1_L8_S2_VP5 C_DIS
;ENDFOLD
TRIGGER WHEN DISTANCE=1 DELAY=-1 DO Schrittmerker_R1Place(10845,10844,FPlace_R1_L8_S2_VP6,XPlace_R1_L8_S2_VP6) PRIO=-1
;FOLD PTP Place_R1_L8_S2_VP6 CONT Vel=12 % PPlace_R1_L8_S2_VP6 Tool[1]:Upper Gripper Base[1]:Rack1;%{PE}%R8.3.21,%MKUKATPBASIS,%CMOVE,%VPTP,%P 1:PTP, 2:Place_R1_L8_S2_VP6, 3:C_DIS, 5:12, 7:PPlace_R1_L8_S2_VP6
$BWDSTART=FALSE
PDAT_ACT= PPPlace_R1_L8_S2_VP6
FDAT_ACT= FPlace_R1_L8_S2_VP6
BAS(#PTP_PARAMS,12)
PTP XPlace_R1_L8_S2_VP6 C_DIS
;ENDFOLD
TRIGGER WHEN DISTANCE=1 DELAY=-1 DO Schrittmerker_R1Place(10846,10845,FPlace_R1_L8_S2_VP7,XPlace_R1_L8_S2_VP7) PRIO=-1
;FOLD PTP Place_R1_L8_S2_VP7 CONT Vel=12 % PPlace_R1_L8_S2_VP7 Tool[1]:Upper Gripper Base[1]:Rack1;%{PE}%R8.3.21,%MKUKATPBASIS,%CMOVE,%VPTP,%P 1:PTP, 2:Place_R1_L8_S2_VP7, 3:C_DIS, 5:12, 7:PPlace_R1_L8_S2_VP7
$BWDSTART=FALSE
PDAT_ACT= PPPlace_R1_L8_S2_VP7
FDAT_ACT= FPlace_R1_L8_S2_VP7
BAS(#PTP_PARAMS,12)
PTP XPlace_R1_L8_S2_VP7 C_DIS
;ENDFOLD

TRIGGER WHEN DISTANCE=1 DELAY=-1 DO Schrittmerker_R1Place(10847,10846,FPlace_R1_L8_S2_Check,XPlace_R1_L8_S2_Check) PRIO=-1
;FOLD PTP Place_R1_L8_S2_Check Vel=12 % PPlace_R1_L8_S2_Check Tool[1]:Upper Gripper Base[1]:Rack1;%{PE}%R8.3.21,%MKUKATPBASIS,%CMOVE,%VPTP,%P 1:PTP, 2:Place_R1_L8_S2_Check, 3:, 5:12, 7:PPlace_R1_L8_S2_Check
$BWDSTART=FALSE
PDAT_ACT= PPPlace_R1_L8_S2_Check
FDAT_ACT= FPlace_R1_L8_S2_Check
BAS(#PTP_PARAMS,12)
PTP XPlace_R1_L8_S2_Check
;ENDFOLD

;***************************************************
;FOLD Pruefe Platz frei
IF (DetectPart(CHECK_SHELF,PLACE)==OCCUPIED) THEN
  UP_Rueckzug_R1Place( )
  RETURN
ENDIF
;ENDFOLD
;***************************************************

TRIGGER WHEN DISTANCE=1 DELAY=-1 DO Schrittmerker_R1Place(10848,10847,FPlace_R1_L8_S2_VP8,XPlace_R1_L8_S2_VP8) PRIO=-1
;FOLD LIN Place_R1_L8_S2_VP8 CONT Vel=0.5 m/s LPlace_R1_L8_S2_VP8 Tool[1]:Upper Gripper Base[1]:Rack1;%{PE}%R8.3.21,%MKUKATPBASIS,%CMOVE,%VLIN,%P 1:LIN, 2:Place_R1_L8_S2_VP8, 3:C_DIS C_DIS, 5:0.5, 7:LPlace_R1_L8_S2_VP8
$BWDSTART=FALSE
LDAT_ACT= LLPlace_R1_L8_S2_VP8
FDAT_ACT= FPlace_R1_L8_S2_VP8
BAS(#CP_PARAMS,0.5)
LIN XPlace_R1_L8_S2_VP8 C_DIS C_DIS
;ENDFOLD

;FOLD Test the way back home - part 1
CONTINUE
IF ($FLAG[M_Test_GrdstFahren1] AND NOT $FLAG[M_Test_GrdstFahren2]) THEN
  $FLAG[M_Test_GrdstFahren2]=TRUE
  UP_Rueckzug( )
  RETURN
ENDIF
;ENDFOLD

;-------------------------------
; Place part position
;-------------------------------
TRIGGER WHEN DISTANCE=1 DELAY=-1 DO Schrittmerker_R1Place(10849,10850,FPlace_R1_L8_S2_AP,XPlace_R1_L8_S2_AP) PRIO=-1
;FOLD LIN Place_R1_L8_S2_AP Vel=0.2 m/s LPlace_R1_L8_S2_AP Tool[1]:Upper Gripper Base[1]:Rack1;%{PE}%R8.3.21,%MKUKATPBASIS,%CMOVE,%VLIN,%P 1:LIN, 2:Place_R1_L8_S2_AP, 3:, 5:0.2, 7:LPlace_R1_L8_S2_AP
$BWDSTART=FALSE
LDAT_ACT= LLPlace_R1_L8_S2_AP
FDAT_ACT= FPlace_R1_L8_S2_AP
BAS(#CP_PARAMS,0.2)
LIN XPlace_R1_L8_S2_AP
;ENDFOLD

;FOLD Test the way back home - part 2
CONTINUE
IF $FLAG[M_Test_GrdstFahren2] THEN
  $FLAG[M_Test_GrdstFahren2]=FALSE
  UP_Rueckzug( )
  RETURN
ENDIF
;ENDFOLD

;***************************************************
; Disable part lost detection
SetPartLostDetection(NO_PART)
;***************************************************

TRIGGER WHEN DISTANCE=1 DELAY=-1 DO Schrittmerker_R1Place(10850,10851,FPlace_R1_L8_S2_NP1,XPlace_R1_L8_S2_NP1) PRIO=-1
;FOLD LIN Place_R1_L8_S2_NP1 Vel=0.2 m/s LPlace_R1_L8_S2_NP1 Tool[1]:Upper Gripper Base[1]:Rack1;%{PE}%R8.3.21,%MKUKATPBASIS,%CMOVE,%VLIN,%P 1:LIN, 2:Place_R1_L8_S2_NP1, 3:C_DIS C_DIS, 5:0.2, 7:LPlace_R1_L8_S2_NP1
$BWDSTART=FALSE
LDAT_ACT= LLPlace_R1_L8_S2_NP1
FDAT_ACT= FPlace_R1_L8_S2_NP1
BAS(#CP_PARAMS,0.2)
LIN XPlace_R1_L8_S2_NP1
;ENDFOLD

;***************************************************
; Check for part present (empty gripper)
CheckPartPresent(EMPTY_GRIPPER)
;***************************************************
; set load data
SetLoadData( )
;***************************************************

TRIGGER WHEN DISTANCE=1 DELAY=-1 DO Schrittmerker_R1Place(10851,10852,FPlace_R1_L8_S2_NP2,XPlace_R1_L8_S2_NP2) PRIO=-1
;FOLD LIN Place_R1_L8_S2_NP2 Vel=0.5 m/s LPlace_R1_L8_S2_NP2 Tool[1]:Upper Gripper Base[1]:Rack1;%{PE}%R8.3.21,%MKUKATPBASIS,%CMOVE,%VLIN,%P 1:LIN, 2:Place_R1_L8_S2_NP2, 3:, 5:0.5, 7:LPlace_R1_L8_S2_NP2
$BWDSTART=FALSE
LDAT_ACT= LLPlace_R1_L8_S2_NP2
FDAT_ACT= FPlace_R1_L8_S2_NP2
BAS(#CP_PARAMS,0.5)
LIN XPlace_R1_L8_S2_NP2
;ENDFOLD
TRIGGER WHEN DISTANCE=1 DELAY=-1 DO Schrittmerker_R1Place(10852,10853,FPlace_R1_L8_S2_NP3,XPlace_R1_L8_S2_NP3) PRIO=-1
;FOLD PTP Place_R1_L8_S2_NP3 CONT Vel=100 % PPlace_R1_L8_S2_NP3 Tool[1]:Upper Gripper Base[0];%{PE}%R8.3.21,%MKUKATPBASIS,%CMOVE,%VPTP,%P 1:PTP, 2:Place_R1_L8_S2_NP3, 3:C_DIS, 5:100, 7:PPlace_R1_L8_S2_NP3
$BWDSTART=FALSE
PDAT_ACT= PPPlace_R1_L8_S2_NP3
FDAT_ACT= FPlace_R1_L8_S2_NP3
BAS(#PTP_PARAMS,100)
PTP XPlace_R1_L8_S2_NP3 C_DIS
;ENDFOLD
TRIGGER WHEN DISTANCE=1 DELAY=-1 DO Schrittmerker_R1Place(10853,10854,FPlace_R1_L8_S2_NP4,XPlace_R1_L8_S2_NP4) PRIO=-1
;FOLD PTP Place_R1_L8_S2_NP4 CONT Vel=100 % PPlace_R1_L8_S2_NP4 Tool[1]:Upper Gripper Base[0];%{PE}%R8.3.21,%MKUKATPBASIS,%CMOVE,%VPTP,%P 1:PTP, 2:Place_R1_L8_S2_NP4, 3:C_DIS, 5:100, 7:PPlace_R1_L8_S2_NP4
$BWDSTART=FALSE
PDAT_ACT= PPPlace_R1_L8_S2_NP4
FDAT_ACT= FPlace_R1_L8_S2_NP4
BAS(#PTP_PARAMS,100)
PTP XPlace_R1_L8_S2_NP4 C_DIS
;ENDFOLD
TRIGGER WHEN DISTANCE=1 DELAY=-1 DO Schrittmerker_R1Place(10854,10855,FPlace_R1_L8_S2_NP5,XPlace_R1_L8_S2_NP5) PRIO=-1
;FOLD PTP Place_R1_L8_S2_NP5 CONT Vel=100 % PPlace_R1_L8_S2_NP5 Tool[1]:Upper Gripper Base[0];%{PE}%R8.3.21,%MKUKATPBASIS,%CMOVE,%VPTP,%P 1:PTP, 2:Place_R1_L8_S2_NP5, 3:C_DIS, 5:100, 7:PPlace_R1_L8_S2_NP5
$BWDSTART=FALSE
PDAT_ACT= PPPlace_R1_L8_S2_NP5
FDAT_ACT= FPlace_R1_L8_S2_NP5
BAS(#PTP_PARAMS,100)
PTP XPlace_R1_L8_S2_NP5 C_DIS
;ENDFOLD

TRIGGER WHEN DISTANCE=1 DELAY=-1 DO Schrittmerker_R1Place(10855,10501,FHOME,$nullframe,XHOME) PRIO=-1
;FOLD PTP HOME Vel=100 % PHome;%{PE}%R8.3.21,%MKUKATPBASIS,%CMOVE,%VPTP,%P 1:PTP, 2:HOME, 3:, 5:100, 7:PHome
$BWDSTART=FALSE
PDAT_ACT= PPHome
FDAT_ACT= FHOME
BAS(#PTP_PARAMS,100)
PTP XHOME
;ENDFOLD

;***************************************************
;FOLD Final tasks.
; Robot out of area Rack 1 Level 8
RobAusStorage1_8_A74=RESET_IN_AREA
;***************************************************
; stop cyclic clearence check
$CYCFLAG[ciFreigabeSPS]=DISABLE_MONITORING
;***************************************************
; Disable collision detection
;FOLD COLLDETECT Off ;%{PE}
;FOLD Parameters ;%{h}
;Params IlfProvider=kukaroboter.basistech.inlineforms.colldetect.off; CollDetect.Command=Off
;ENDFOLD
USE_CD_PARAMS(0)
;ENDFOLD
;***************************************************
;ENDFOLD
;***************************************************

END

; ##################################################

GLOBAL DEF UP_Place_R1_L8_S3( )
;***************************************************
; Place part on:
;    Rack  1
;    Level 8
;    Shelf 3
;***************************************************
;FOLD Preconditions - Vorraussetzungen
;***************************************************
; Enable collision detection
;FOLD COLLDETECT SetLimits Axis1: 150 % Axis2: 200 % Axis3: 150 % Axis4: 200 % Axis5: 150 % Axis6: 150 % ;%{PE}
;FOLD Parameters ;%{h}
;Params IlfProvider=kukaroboter.basistech.inlineforms.colldetect.setlimits; CollDetect.Command=SetLimits; CollDetect.Axis1=150; CollDetect.Axis2=200; CollDetect.Axis3=150; CollDetect.Axis4=200; CollDetect.Axis5=150; CollDetect.Axis6=150
;ENDFOLD
SET_TQ_VALUES(150, 200, 150, 200, 150, 150)
;ENDFOLD
;***************************************************
; Check for part in gripper (tool 1).
CheckPartPresent(OCCUPIED_GRIPPER,PART_ON_TOOL_1)
;***************************************************
; Enable part lost detection for tool 1
SetPartLostDetection(PART_ON_TOOL_1)
;***************************************************
; Set load data.
SetLoadData( )
;***************************************************
; Robot has to start from home position.
IF NOT $IN_HOME THEN
  UP_HomeToHome(0)
ENDIF
;***************************************************
;ENDFOLD

TRIGGER WHEN DISTANCE=1 DELAY=-1 DO Schrittmerker_R1Place(10501,10501,FHOME,$nullframe,XHOME) PRIO=-1
;FOLD PTP HOME Vel=12 % PHome;%{PE}%R8.3.21,%MKUKATPBASIS,%CMOVE,%VPTP,%P 1:PTP, 2:HOME, 3:, 5:12, 7:PHome
$BWDSTART=FALSE
PDAT_ACT= PPHome
FDAT_ACT= FHOME
BAS(#PTP_PARAMS,12)
PTP XHOME
;ENDFOLD

;***************************************************
;FOLD Area clearence handshake.
IF NOT $FLAG[M_Inbetriebnahme] THEN
  ;-------------------------------------------------
  ; Request area clearence.
  AnfStoer_Store1_8_A106=SET_REQUEST
  ;-------------------------------------------------
  ; Wait for area clearence from PLC.
  WAIT_FOR_INPUT("Frg_Storage1_8_E74",TRUE)
  ;-------------------------------------------------
  ; Reset area clearence request.
  AnfStoer_Store1_8_A106=RESET_REQUEST
  ;-------------------------------------------------
  ; start cyclic clearence check
  $CYCFLAG[ciFreigabeSPS]=Frg_Storage1_8_E74
  ;-------------------------------------------------
ENDIF
;***************************************************
; set "robot in area"
RobAusStorage1_8_A74=SET_IN_AREA
;ENDFOLD
;***************************************************

;***************************************************
;FOLD Check for Teachmode
IF $FLAG[M_Teachen] THEN
  WAIT FOR $T1
ENDIF
;ENDFOLD
;***************************************************

; move to the rack
TRIGGER WHEN DISTANCE=1 DELAY=-1 DO Schrittmerker_R1Place(10860,10501,FPlace_R1_L8_S3_VP1,XPlace_R1_L8_S3_VP1) PRIO=-1
;FOLD PTP Place_R1_L8_S3_VP1 CONT Vel=12 % PPlace_R1_L8_S3_VP1 Tool[1]:Upper Gripper Base[0];%{PE}%R8.3.21,%MKUKATPBASIS,%CMOVE,%VPTP,%P 1:PTP, 2:Place_R1_L8_S3_VP1, 3:C_DIS, 5:12, 7:PPlace_R1_L8_S3_VP1
$BWDSTART=FALSE
PDAT_ACT= PPPlace_R1_L8_S3_VP1
FDAT_ACT= FPlace_R1_L8_S3_VP1
BAS(#PTP_PARAMS,12)
PTP XPlace_R1_L8_S3_VP1 C_DIS
;ENDFOLD
TRIGGER WHEN DISTANCE=1 DELAY=-1 DO Schrittmerker_R1Place(10861,10860,FPlace_R1_L8_S3_VP2,XPlace_R1_L8_S3_VP2) PRIO=-1
;FOLD PTP Place_R1_L8_S3_VP2 CONT Vel=12 % PPlace_R1_L8_S3_VP2 Tool[1]:Upper Gripper Base[0];%{PE}%R8.3.21,%MKUKATPBASIS,%CMOVE,%VPTP,%P 1:PTP, 2:Place_R1_L8_S3_VP2, 3:C_DIS, 5:12, 7:PPlace_R1_L8_S3_VP2
$BWDSTART=FALSE
PDAT_ACT= PPPlace_R1_L8_S3_VP2
FDAT_ACT= FPlace_R1_L8_S3_VP2
BAS(#PTP_PARAMS,12)
PTP XPlace_R1_L8_S3_VP2 C_DIS
;ENDFOLD
TRIGGER WHEN DISTANCE=1 DELAY=-1 DO Schrittmerker_R1Place(10862,10861,FPlace_R1_L8_S3_VP3,XPlace_R1_L8_S3_VP3) PRIO=-1
;FOLD PTP Place_R1_L8_S3_VP3 CONT Vel=12 % PPlace_R1_L8_S3_VP3 Tool[1]:Upper Gripper Base[0];%{PE}%R8.3.21,%MKUKATPBASIS,%CMOVE,%VPTP,%P 1:PTP, 2:Place_R1_L8_S3_VP3, 3:C_DIS, 5:12, 7:PPlace_R1_L8_S3_VP3
$BWDSTART=FALSE
PDAT_ACT= PPPlace_R1_L8_S3_VP3
FDAT_ACT= FPlace_R1_L8_S3_VP3
BAS(#PTP_PARAMS,12)
PTP XPlace_R1_L8_S3_VP3 C_DIS
;ENDFOLD
TRIGGER WHEN DISTANCE=1 DELAY=-1 DO Schrittmerker_R1Place(10863,10862,FPlace_R1_L8_S3_VP4,XPlace_R1_L8_S3_VP4) PRIO=-1
;FOLD PTP Place_R1_L8_S3_VP4 CONT Vel=12 % PPlace_R1_L8_S3_VP4 Tool[1]:Upper Gripper Base[0];%{PE}%R8.3.21,%MKUKATPBASIS,%CMOVE,%VPTP,%P 1:PTP, 2:Place_R1_L8_S3_VP4, 3:C_DIS, 5:12, 7:PPlace_R1_L8_S3_VP4
$BWDSTART=FALSE
PDAT_ACT= PPPlace_R1_L8_S3_VP4
FDAT_ACT= FPlace_R1_L8_S3_VP4
BAS(#PTP_PARAMS,12)
PTP XPlace_R1_L8_S3_VP4 C_DIS
;ENDFOLD
TRIGGER WHEN DISTANCE=1 DELAY=-1 DO Schrittmerker_R1Place(10864,10863,FPlace_R1_L8_S3_VP5,XPlace_R1_L8_S3_VP5) PRIO=-1
;FOLD PTP Place_R1_L8_S3_VP5 CONT Vel=12 % PPlace_R1_L8_S3_VP5 Tool[1]:Upper Gripper Base[0];%{PE}%R8.3.21,%MKUKATPBASIS,%CMOVE,%VPTP,%P 1:PTP, 2:Place_R1_L8_S3_VP5, 3:C_DIS, 5:12, 7:PPlace_R1_L8_S3_VP5
$BWDSTART=FALSE
PDAT_ACT= PPPlace_R1_L8_S3_VP5
FDAT_ACT= FPlace_R1_L8_S3_VP5
BAS(#PTP_PARAMS,12)
PTP XPlace_R1_L8_S3_VP5 C_DIS
;ENDFOLD

TRIGGER WHEN DISTANCE=1 DELAY=-1 DO Schrittmerker_R1Place(10865,10864,FPlace_R1_L8_S3_Check,XPlace_R1_L8_S3_Check) PRIO=-1
;FOLD PTP Place_R1_L8_S3_Check Vel=12 % PPlace_R1_L8_S3_Check Tool[1]:Upper Gripper Base[1]:Rack1;%{PE}%R8.3.21,%MKUKATPBASIS,%CMOVE,%VPTP,%P 1:PTP, 2:Place_R1_L8_S3_Check, 3:, 5:12, 7:PPlace_R1_L8_S3_Check
$BWDSTART=FALSE
PDAT_ACT= PPPlace_R1_L8_S3_Check
FDAT_ACT= FPlace_R1_L8_S3_Check
BAS(#PTP_PARAMS,12)
PTP XPlace_R1_L8_S3_Check
;ENDFOLD

;***************************************************
;FOLD Pruefe Platz frei
IF (DetectPart(CHECK_SHELF,PLACE)==OCCUPIED) THEN
  UP_Rueckzug_R1Place( )
  RETURN
ENDIF
;ENDFOLD
;***************************************************

TRIGGER WHEN DISTANCE=1 DELAY=-1 DO Schrittmerker_R1Place(10866,10865,FPlace_R1_L8_S3_VP6,XPlace_R1_L8_S3_VP6) PRIO=-1
;FOLD LIN Place_R1_L8_S3_VP6 CONT Vel=0.5 m/s LPlace_R1_L8_S3_VP6 Tool[1]:Upper Gripper Base[1]:Rack1;%{PE}%R8.3.21,%MKUKATPBASIS,%CMOVE,%VLIN,%P 1:LIN, 2:Place_R1_L8_S3_VP6, 3:C_DIS C_DIS, 5:0.5, 7:LPlace_R1_L8_S3_VP6
$BWDSTART=FALSE
LDAT_ACT= LLPlace_R1_L8_S3_VP6
FDAT_ACT= FPlace_R1_L8_S3_VP6
BAS(#CP_PARAMS,0.5)
LIN XPlace_R1_L8_S3_VP6 C_DIS C_DIS
;ENDFOLD
TRIGGER WHEN DISTANCE=1 DELAY=-1 DO Schrittmerker_R1Place(10867,10866,FPlace_R1_L8_S3_VP7,XPlace_R1_L8_S3_VP7) PRIO=-1
;FOLD LIN Place_R1_L8_S3_VP7 CONT Vel=0.5 m/s LPlace_R1_L8_S3_VP7 Tool[1]:Upper Gripper Base[1]:Rack1;%{PE}%R8.3.21,%MKUKATPBASIS,%CMOVE,%VLIN,%P 1:LIN, 2:Place_R1_L8_S3_VP7, 3:C_DIS C_DIS, 5:0.5, 7:LPlace_R1_L8_S3_VP7
$BWDSTART=FALSE
LDAT_ACT= LLPlace_R1_L8_S3_VP7
FDAT_ACT= FPlace_R1_L8_S3_VP7
BAS(#CP_PARAMS,0.5)
LIN XPlace_R1_L8_S3_VP7 C_DIS C_DIS
;ENDFOLD
TRIGGER WHEN DISTANCE=1 DELAY=-1 DO Schrittmerker_R1Place(10868,10867,FPlace_R1_L8_S3_VP8,XPlace_R1_L8_S3_VP8) PRIO=-1
;FOLD LIN Place_R1_L8_S3_VP8 CONT Vel=0.5 m/s LPlace_R1_L8_S3_VP8 Tool[1]:Upper Gripper Base[1]:Rack1;%{PE}%R8.3.21,%MKUKATPBASIS,%CMOVE,%VLIN,%P 1:LIN, 2:Place_R1_L8_S3_VP8, 3:C_DIS C_DIS, 5:0.5, 7:LPlace_R1_L8_S3_VP8
$BWDSTART=FALSE
LDAT_ACT= LLPlace_R1_L8_S3_VP8
FDAT_ACT= FPlace_R1_L8_S3_VP8
BAS(#CP_PARAMS,0.5)
LIN XPlace_R1_L8_S3_VP8 C_DIS C_DIS
;ENDFOLD

;FOLD Test the way back home - part 1
CONTINUE
IF ($FLAG[M_Test_GrdstFahren1] AND NOT $FLAG[M_Test_GrdstFahren2]) THEN
  $FLAG[M_Test_GrdstFahren2]=TRUE
  UP_Rueckzug( )
  RETURN
ENDIF
;ENDFOLD

;-------------------------------
; Place part position
;-------------------------------
TRIGGER WHEN DISTANCE=1 DELAY=-1 DO Schrittmerker_R1Place(10869,10870,FPlace_R1_L8_S3_AP,XPlace_R1_L8_S3_AP) PRIO=-1
;FOLD LIN Place_R1_L8_S3_AP Vel=0.2 m/s LPlace_R1_L8_S3_AP Tool[1]:Upper Gripper Base[1]:Rack1;%{PE}%R8.3.21,%MKUKATPBASIS,%CMOVE,%VLIN,%P 1:LIN, 2:Place_R1_L8_S3_AP, 3:, 5:0.2, 7:LPlace_R1_L8_S3_AP
$BWDSTART=FALSE
LDAT_ACT= LLPlace_R1_L8_S3_AP
FDAT_ACT= FPlace_R1_L8_S3_AP
BAS(#CP_PARAMS,0.2)
LIN XPlace_R1_L8_S3_AP
;ENDFOLD

;FOLD Test the way back home - part 2
CONTINUE
IF $FLAG[M_Test_GrdstFahren2] THEN
  $FLAG[M_Test_GrdstFahren2]=FALSE
  UP_Rueckzug( )
  RETURN
ENDIF
;ENDFOLD

;***************************************************
; Disable part lost detection
SetPartLostDetection(NO_PART)
;***************************************************

TRIGGER WHEN DISTANCE=1 DELAY=-1 DO Schrittmerker_R1Place(10870,10871,FPlace_R1_L8_S3_NP1,XPlace_R1_L8_S3_NP1) PRIO=-1
;FOLD LIN Place_R1_L8_S3_NP1 Vel=0.2 m/s LPlace_R1_L8_S3_NP1 Tool[1]:Upper Gripper Base[1]:Rack1;%{PE}%R8.3.21,%MKUKATPBASIS,%CMOVE,%VLIN,%P 1:LIN, 2:Place_R1_L8_S3_NP1, 3:C_DIS C_DIS, 5:0.2, 7:LPlace_R1_L8_S3_NP1
$BWDSTART=FALSE
LDAT_ACT= LLPlace_R1_L8_S3_NP1
FDAT_ACT= FPlace_R1_L8_S3_NP1
BAS(#CP_PARAMS,0.2)
LIN XPlace_R1_L8_S3_NP1
;ENDFOLD

;***************************************************
; Check for part present (empty gripper)
CheckPartPresent(EMPTY_GRIPPER)
;***************************************************
; set load data
SetLoadData( )
;***************************************************

TRIGGER WHEN DISTANCE=1 DELAY=-1 DO Schrittmerker_R1Place(10871,10872,FPlace_R1_L8_S3_NP2,XPlace_R1_L8_S3_NP2) PRIO=-1
;FOLD LIN Place_R1_L8_S3_NP2 Vel=0.5 m/s LPlace_R1_L8_S3_NP2 Tool[1]:Upper Gripper Base[1]:Rack1;%{PE}%R8.3.21,%MKUKATPBASIS,%CMOVE,%VLIN,%P 1:LIN, 2:Place_R1_L8_S3_NP2, 3:, 5:0.5, 7:LPlace_R1_L8_S3_NP2
$BWDSTART=FALSE
LDAT_ACT= LLPlace_R1_L8_S3_NP2
FDAT_ACT= FPlace_R1_L8_S3_NP2
BAS(#CP_PARAMS,0.5)
LIN XPlace_R1_L8_S3_NP2
;ENDFOLD
TRIGGER WHEN DISTANCE=1 DELAY=-1 DO Schrittmerker_R1Place(10872,10873,FPlace_R1_L8_S3_NP3,XPlace_R1_L8_S3_NP3) PRIO=-1
;FOLD PTP Place_R1_L8_S3_NP3 CONT Vel=100 % PPlace_R1_L8_S3_NP3 Tool[1]:Upper Gripper Base[0];%{PE}%R8.3.21,%MKUKATPBASIS,%CMOVE,%VPTP,%P 1:PTP, 2:Place_R1_L8_S3_NP3, 3:C_DIS, 5:100, 7:PPlace_R1_L8_S3_NP3
$BWDSTART=FALSE
PDAT_ACT= PPPlace_R1_L8_S3_NP3
FDAT_ACT= FPlace_R1_L8_S3_NP3
BAS(#PTP_PARAMS,100)
PTP XPlace_R1_L8_S3_NP3 C_DIS
;ENDFOLD
TRIGGER WHEN DISTANCE=1 DELAY=-1 DO Schrittmerker_R1Place(10873,10874,FPlace_R1_L8_S3_NP4,XPlace_R1_L8_S3_NP4) PRIO=-1
;FOLD PTP Place_R1_L8_S3_NP4 CONT Vel=100 % PPlace_R1_L8_S3_NP4 Tool[1]:Upper Gripper Base[0];%{PE}%R8.3.21,%MKUKATPBASIS,%CMOVE,%VPTP,%P 1:PTP, 2:Place_R1_L8_S3_NP4, 3:C_DIS, 5:100, 7:PPlace_R1_L8_S3_NP4
$BWDSTART=FALSE
PDAT_ACT= PPPlace_R1_L8_S3_NP4
FDAT_ACT= FPlace_R1_L8_S3_NP4
BAS(#PTP_PARAMS,100)
PTP XPlace_R1_L8_S3_NP4 C_DIS
;ENDFOLD

TRIGGER WHEN DISTANCE=1 DELAY=-1 DO Schrittmerker_R1Place(10874,10501,FHOME,$nullframe,XHOME) PRIO=-1
;FOLD PTP HOME Vel=100 % PHome;%{PE}%R8.3.21,%MKUKATPBASIS,%CMOVE,%VPTP,%P 1:PTP, 2:HOME, 3:, 5:100, 7:PHome
$BWDSTART=FALSE
PDAT_ACT= PPHome
FDAT_ACT= FHOME
BAS(#PTP_PARAMS,100)
PTP XHOME
;ENDFOLD

;***************************************************
;FOLD Final tasks.
; Robot out of area Rack 1 Level 8
RobAusStorage1_8_A74=RESET_IN_AREA
;***************************************************
; stop cyclic clearence check
$CYCFLAG[ciFreigabeSPS]=DISABLE_MONITORING
;***************************************************
; Disable collision detection
;FOLD COLLDETECT Off ;%{PE}
;FOLD Parameters ;%{h}
;Params IlfProvider=kukaroboter.basistech.inlineforms.colldetect.off; CollDetect.Command=Off
;ENDFOLD
USE_CD_PARAMS(0)
;ENDFOLD
;***************************************************
;ENDFOLD
;***************************************************

END

; ##################################################

GLOBAL DEF UP_Place_R1_L8_S4( )
;***************************************************
; Place part on:
;    Rack  1
;    Level 8
;    Shelf 4
;***************************************************
;FOLD Preconditions - Vorraussetzungen
;***************************************************
; Enable collision detection
;FOLD COLLDETECT SetLimits Axis1: 150 % Axis2: 200 % Axis3: 150 % Axis4: 200 % Axis5: 150 % Axis6: 150 % ;%{PE}
;FOLD Parameters ;%{h}
;Params IlfProvider=kukaroboter.basistech.inlineforms.colldetect.setlimits; CollDetect.Command=SetLimits; CollDetect.Axis1=150; CollDetect.Axis2=200; CollDetect.Axis3=150; CollDetect.Axis4=200; CollDetect.Axis5=150; CollDetect.Axis6=150
;ENDFOLD
SET_TQ_VALUES(150, 200, 150, 200, 150, 150)
;ENDFOLD
;***************************************************
; Check for part in gripper (tool 1).
CheckPartPresent(OCCUPIED_GRIPPER,PART_ON_TOOL_1)
;***************************************************
; Enable part lost detection for tool 1
SetPartLostDetection(PART_ON_TOOL_1)
;***************************************************
; Set load data.
SetLoadData( )
;***************************************************
; Robot has to start from home position.
IF NOT $IN_HOME THEN
  UP_HomeToHome(0)
ENDIF
;***************************************************
;ENDFOLD

TRIGGER WHEN DISTANCE=1 DELAY=-1 DO Schrittmerker_R1Place(10501,10501,FHOME,$nullframe,XHOME) PRIO=-1
;FOLD PTP HOME Vel=12 % PHome;%{PE}%R8.3.21,%MKUKATPBASIS,%CMOVE,%VPTP,%P 1:PTP, 2:HOME, 3:, 5:12, 7:PHome
$BWDSTART=FALSE
PDAT_ACT= PPHome
FDAT_ACT= FHOME
BAS(#PTP_PARAMS,12)
PTP XHOME
;ENDFOLD

;***************************************************
;FOLD Area clearence handshake.
IF NOT $FLAG[M_Inbetriebnahme] THEN
  ;-------------------------------------------------
  ; Request area clearence.
  AnfStoer_Store1_8_A106=SET_REQUEST
  ;-------------------------------------------------
  ; Wait for area clearence from PLC.
  WAIT_FOR_INPUT("Frg_Storage1_8_E74",TRUE)
  ;-------------------------------------------------
  ; Reset area clearence request.
  AnfStoer_Store1_8_A106=RESET_REQUEST
  ;-------------------------------------------------
  ; start cyclic clearence check
  $CYCFLAG[ciFreigabeSPS]=Frg_Storage1_8_E74
  ;-------------------------------------------------
ENDIF
;***************************************************
; set "robot in area"
RobAusStorage1_8_A74=SET_IN_AREA
;ENDFOLD
;***************************************************

;***************************************************
;FOLD Check for Teachmode
IF $FLAG[M_Teachen] THEN
  WAIT FOR $T1
ENDIF
;ENDFOLD
;***************************************************

